# B&R Automation Studio project EFI (part 7)

### IOMap.iom - PC_any/IOMap.iom
```iecst
(********************************************************************
 * COPYRIGHT -- Bernecker + Rainer
 ********************************************************************
 * File: IoMap.iom
 * Author: B+R
 ********************************************************************
 * IO mapping file
 ********************************************************************)
VAR_CONFIG
	Cyclic#1.::gAxisStepper[1].DrvIf.iLifeCnt AT %IB."X67SM2436".LifeCnt;
	Cyclic#1.::gAxisStepper[1].DrvIf.iDrvOK AT %IX."X67SM2436".DrvOk01;
	Cyclic#1.::gAxisStepper[1].DrvIf.oBoostCurrent AT %QX."X67SM2436".BoostCurrent01;
	Cyclic#1.::gAxisStepper[1].DrvIf.oStandStillCurrent AT %QX."X67SM2436".StandstillCurrent01;
	Cyclic#1.::gAxisStepper[1].DrvIf.oSetTime AT %QW."X67SM2436".SetTime01;
	Cyclic#1.::gAxisStepper[1].MotorStep0 AT %QW."X67SM2436".Motor1Step0;
	Cyclic#1.::gAxisStepper[1].DiDoIf.iLifeCntDriveEnable AT %IB."X67SM2436".LifeCnt;
	Cyclic#1.::gAxisStepper[1].DiDoIf.iLifeCntDriveReady AT %IB."X67SM2436".LifeCnt;
	Cyclic#1.::gAxisStepper[1].DiDoIf.iDriveReady AT %IX."X67SM2436".DrvOk01;
	Cyclic#1.::gAxisStepper[1].DiDoIf.oDriveEnable AT %QX."X67SM2436".DriveEnable01;
	Cyclic#1.::gAxisStepper[1].EncIf1.iLifeCnt AT %IB."X67SM2436".LifeCnt;
	Cyclic#1.::gAxisStepper[1].EncIf1.iEncOK AT %IX."X67SM2436".EncOk01;
	Cyclic#1.::gAxisStepper[1].EncIf1.iActPos AT %IW."X67SM2436".ActPos01;
	Cyclic#1.::gAxisStepper[1].EncIf1.iRefPulsePos AT %IW."X67SM2436".RefPulsePos01;
	Cyclic#1.::gAxisStepper[1].EncIf1.iRefPulseCnt AT %IB."X67SM2436".RefPulseCnt01;
	Cyclic#1.::gAxisStepper[1].EncIf1.iActTime AT %IW."X67SM2436".ActTime01;
	Cyclic#1.::gAxisStepper[2].DrvIf.iLifeCnt AT %IB."X67SM2436".LifeCnt;
	Cyclic#1.::gAxisStepper[2].DrvIf.iDrvOK AT %IX."X67SM2436".DrvOk02;
	Cyclic#1.::gAxisStepper[2].DrvIf.oBoostCurrent AT %QX."X67SM2436".BoostCurrent02;
	Cyclic#1.::gAxisStepper[2].DrvIf.oStandStillCurrent AT %QX."X67SM2436".StandstillCurrent02;
	Cyclic#1.::gAxisStepper[2].DrvIf.oSetTime AT %QW."X67SM2436".SetTime02;
	Cyclic#1.::gAxisStepper[2].MotorStep0 AT %QW."X67SM2436".Motor2Step0;
	Cyclic#1.::gAxisStepper[2].DiDoIf.iLifeCntDriveEnable AT %IB."X67SM2436".LifeCnt;
	Cyclic#1.::gAxisStepper[2].DiDoIf.iLifeCntDriveReady AT %IB."X67SM2436".LifeCnt;
	Cyclic#1.::gAxisStepper[2].DiDoIf.iDriveReady AT %IX."X67SM2436".DrvOk02;
	Cyclic#1.::gAxisStepper[2].DiDoIf.oDriveEnable AT %QX."X67SM2436".DriveEnable02;
	Cyclic#1.::gAxisStepper[2].EncIf1.iLifeCnt AT %IB."X67SM2436".LifeCnt;
	Cyclic#1.::gAxisStepper[2].EncIf1.iEncOK AT %IX."X67SM2436".EncOk02;
	Cyclic#1.::gAxisStepper[2].EncIf1.iActPos AT %IW."X67SM2436".ActPos02;
	Cyclic#1.::gAxisStepper[2].EncIf1.iRefPulsePos AT %IW."X67SM2436".RefPulsePos02;
	Cyclic#1.::gAxisStepper[2].EncIf1.iRefPulseCnt AT %IB."X67SM2436".RefPulseCnt02;
	Cyclic#1.::gAxisStepper[2].EncIf1.iActTime AT %IW."X67SM2436".ActTime02;
	Cyclic#1.::gInverterSignalsPowerLink[1].In.StatusWord AT %IW."8I66xxxxxxx.0P-xxx1".ETAD_Input;
	Cyclic#1.::gInverterSignalsPowerLink[1].In.ActualSpeed AT %IW."8I66xxxxxxx.0P-xxx1".RFRD_Input;
	Cyclic#1.::gInverterSignalsPowerLink[1].In.ErrorID AT %IW."8I66xxxxxxx.0P-xxx1".LFT_Input;
	Cyclic#1.::gInverterSignalsPowerLink[1].Out.ControlWord AT %QW."8I66xxxxxxx.0P-xxx1".CMDD_Output;
	Cyclic#1.::gInverterSignalsPowerLink[1].Out.SetSpeed AT %QW."8I66xxxxxxx.0P-xxx1".LFRD_Output;
	Cyclic#1.::gInverterSignalsPowerLink[1].In.ActualCurrent AT %IW."8I66xxxxxxx.0P-xxx1".LCR_Input;
	Cyclic#1.::gInverterSignalsPowerLink[1].In.DigitalInput[0] AT %IX."8I66xxxxxxx.0P-xxx1".IL1R_Input_DI1;
	Cyclic#1.::gInverterSignalsPowerLink[1].In.DigitalInput[1] AT %IX."8I66xxxxxxx.0P-xxx1".IL1R_Input_DI2;
	Cyclic#1.::gInverterSignalsPowerLink[1].In.DigitalInput[2] AT %IX."8I66xxxxxxx.0P-xxx1".IL1R_Input_DI3;
	Cyclic#1.::gInverterSignalsPowerLink[1].In.DigitalInput[3] AT %IX."8I66xxxxxxx.0P-xxx1".IL1R_Input_DI4;
	Cyclic#1.::gInverterSignalsPowerLink[1].In.DigitalInput[4] AT %IX."8I66xxxxxxx.0P-xxx1".IL1R_Input_DI5;
	Cyclic#1.::gInverterSignalsPowerLink[1].In.DigitalInput[5] AT %IX."8I66xxxxxxx.0P-xxx1".IL1R_Input_DI6;
	Cyclic#1.::gInverterSignalsPowerLink[1].In.DigitalInput[6] AT %IX."8I66xxxxxxx.0P-xxx1".IL1R_Input_DAI1;
	Cyclic#1.::gInverterSignalsPowerLink[1].In.DigitalInput[7] AT %IX."8I66xxxxxxx.0P-xxx1".IL1R_Input_DAI2;
	Cyclic#1.::gInverterSignalsPowerLink[1].In.AnalogInput[0] AT %IW."8I66xxxxxxx.0P-xxx1".AI1R_Input;
	Cyclic#1.::gInverterSignalsPowerLink[1].In.AnalogInput[1] AT %IW."8I66xxxxxxx.0P-xxx1".AI2R_Input;
	Cyclic#1.::gInverterSignalsPowerLink[1].In.AnalogInput[2] AT %IW."8I66xxxxxxx.0P-xxx1".AI3R_Input;
	Cyclic#1.::gInverterSignalsPowerLink[1].Out.AnalogOutput AT %QW."8I66xxxxxxx.0P-xxx1".AO1R_Output;
	Cyclic#1.::gInverterSignalsPowerLink[1].Out.DigitalOutput[0] AT %QX."8I66xxxxxxx.0P-xxx1".OL1R_Output_R1;
	Cyclic#1.::gInverterSignalsPowerLink[1].Out.DigitalOutput[1] AT %QX."8I66xxxxxxx.0P-xxx1".OL1R_Output_R2;
	Cyclic#1.::gInverterSignalsPowerLink[1].Out.DigitalOutput[2] AT %QX."8I66xxxxxxx.0P-xxx1".OL1R_Output_DQ1;
	Cyclic#1.::gInverterSignalsPowerLink[1].In.ActualTorque AT %IW."8I66xxxxxxx.0P-xxx1".OTRN_Input;
	gToWriteDataModbFeeder[1] AT %QW."ModbusFeeder".writeFeederBk2_1;
	gToWriteDataModbFeeder[2] AT %QW."ModbusFeeder".writeFeederBk2_2;
	gToWriteDataModbFeeder[3] AT %QW."ModbusFeeder".writeFeederBk2_3;
	gToWriteDataModbFeeder[4] AT %QW."ModbusFeeder".writeFeederBk2_4;
	gToWriteDataModbFeeder[5] AT %QX."ModbusFeeder".writeFeederBk2_5;
	gToWriteDataModbFeeder[6] AT %QX."ModbusFeeder".writeFeederBk2_6;
	gToWriteDataModbFeeder[7] AT %QX."ModbusFeeder".writeFeederBk2_7;
	gToWriteDataModbFeeder[8] AT %QX."ModbusFeeder".writeFeederBk2_8;
	gToWriteDataModbFeeder[9] AT %QX."ModbusFeeder".writeFeederBk2_9;
	gToWriteDataModbFeeder[10] AT %QX."ModbusFeeder".writeFeederBk2_10;
	gToWriteDataModbFeeder[11] AT %QX."ModbusFeeder".writeFeederBk2_11;
	gToWriteDataModbFeeder[12] AT %QX."ModbusFeeder".writeFeederBk2_12;
	gToWriteDataModbFeeder[13] AT %QX."ModbusFeeder".writeFeederBk2_13;
	gToWriteDataModbFeeder[14] AT %QX."ModbusFeeder".writeFeederBk2_14;
	gToWriteDataModbFeeder[15] AT %QX."ModbusFeeder".writeFeederBk2_15;
	gToWriteDataModbFeeder[16] AT %QX."ModbusFeeder".writeFeederBk2_16;
	gToWriteDataModbFeeder[17] AT %QX."ModbusFeeder".writeFeederBk2_17;
	gToWriteDataModbFeeder[18] AT %QX."ModbusFeeder".writeFeederBk2_18;
	gToWriteDataModbFeeder[19] AT %QX."ModbusFeeder".writeFeederBk2_19;
	gToWriteDataModbFeeder[20] AT %QX."ModbusFeeder".writeFeederBk2_20;
	gToWriteDataModbFeeder[21] AT %QX."ModbusFeeder".writeFeederBk2_21;
	gToWriteDataModbFeeder[22] AT %QX."ModbusFeeder".writeFeederBk2_22;
	gToWriteDataModbFeeder[23] AT %QX."ModbusFeeder".writeFeederBk2_23;
	gToWriteDataModbFeeder[24] AT %QX."ModbusFeeder".writeFeederBk2_24;
	gToWriteDataModbFeeder[25] AT %QX."ModbusFeeder".writeFeederBk2_25;
	gReceivedDataModbFeeder[1] AT %IW."ModbusFeeder".readFeederBk1_1;
	gReceivedDataModbFeeder[2] AT %IW."ModbusFeeder".readFeederBk1_2;
	gReceivedDataModbFeeder[3] AT %IW."ModbusFeeder".readFeederBk1_3;
	gReceivedDataModbFeeder[4] AT %IW."ModbusFeeder".readFeederBk1_4;
	gToWriteDataModbFeeder[5] AT %IX."ModbusFeeder".readFeederBk1_5;
	gToWriteDataModbFeeder[6] AT %IX."ModbusFeeder".readFeederBk1_6;
	gToWriteDataModbFeeder[7] AT %IX."ModbusFeeder".readFeederBk1_7;
	gToWriteDataModbFeeder[8] AT %IX."ModbusFeeder".readFeederBk1_8;
	gToWriteDataModbFeeder[9] AT %IX."ModbusFeeder".readFeederBk1_9;
	gToWriteDataModbFeeder[10] AT %IX."ModbusFeeder".readFeederBk1_10;
	gToWriteDataModbFeeder[11] AT %IX."ModbusFeeder".readFeederBk1_11;
	gToWriteDataModbFeeder[12] AT %IX."ModbusFeeder".readFeederBk1_12;
	gToWriteDataModbFeeder[13] AT %IX."ModbusFeeder".readFeederBk1_13;
	gToWriteDataModbFeeder[14] AT %IX."ModbusFeeder".readFeederBk1_14;
	gToWriteDataModbFeeder[15] AT %IX."ModbusFeeder".readFeederBk1_15;
	gToWriteDataModbFeeder[16] AT %IX."ModbusFeeder".readFeederBk1_16;
	gToWriteDataModbFeeder[17] AT %IX."ModbusFeeder".readFeederBk1_17;
	gToWriteDataModbFeeder[18] AT %IX."ModbusFeeder".readFeederBk1_18;
	gToWriteDataModbFeeder[19] AT %IX."ModbusFeeder".readFeederBk1_19;
	gToWriteDataModbFeeder[20] AT %IX."ModbusFeeder".readFeederBk1_20;
	gToWriteDataModbFeeder[21] AT %IX."ModbusFeeder".readFeederBk1_21;
	gToWriteDataModbFeeder[22] AT %IX."ModbusFeeder".readFeederBk1_22;
	gToWriteDataModbFeeder[23] AT %IX."ModbusFeeder".readFeederBk1_23;
	gToWriteDataModbFeeder[24] AT %IX."ModbusFeeder".readFeederBk1_24;
	gToWriteDataModbFeeder[25] AT %IX."ModbusFeeder".readFeederBk1_25;
	gToWriteDataModbCoater[1] AT %QW."ModbusPrimer".writeCoaterBk2_1;
	gToWriteDataModbCoater[2] AT %QW."ModbusPrimer".writeCoaterBk2_2;
	gToWriteDataModbCoater[3] AT %QW."ModbusPrimer".writeCoaterBk2_3;
	gToWriteDataModbCoater[4] AT %QW."ModbusPrimer".writeCoaterBk2_4;
	gToWriteDataModbCoater[5] AT %QW."ModbusPrimer".writeCoaterBk2_5;
	gToWriteDataModbCoater[6] AT %QW."ModbusPrimer".writeCoaterBk2_6;
	gToWriteDataModbCoater[7] AT %QW."ModbusPrimer".writeCoaterBk2_7;
	gToWriteDataModbCoater[8] AT %QW."ModbusPrimer".writeCoaterBk2_8;
	gToWriteDataModbCoater[9] AT %QW."ModbusPrimer".writeCoaterBk2_9;
	gToWriteDataModbCoater[10] AT %QW."ModbusPrimer".writeCoaterBk2_10;
	gToWriteDataModbCoater[11] AT %QW."ModbusPrimer".writeCoaterBk2_11;
	gToWriteDataModbCoater[12] AT %QW."ModbusPrimer".writeCoaterBk2_12;
	gToWriteDataModbCoater[13] AT %QW."ModbusPrimer".writeCoaterBk2_13;
	gToWriteDataModbCoater[14] AT %QW."ModbusPrimer".writeCoaterBk2_14;
	gToWriteDataModbCoater[15] AT %QW."ModbusPrimer".writeCoaterBk2_15;
	gToWriteDataModbCoater[16] AT %QW."ModbusPrimer".writeCoaterBk2_16;
	gToWriteDataModbCoater[17] AT %QW."ModbusPrimer".writeCoaterBk2_17;
	gToWriteDataModbCoater[18] AT %QW."ModbusPrimer".writeCoaterBk2_18;
	gToWriteDataModbCoater[19] AT %QW."ModbusPrimer".writeCoaterBk2_19;
	gToWriteDataModbCoater[20] AT %QW."ModbusPrimer".writeCoaterBk2_20;
	gToWriteDataModbCoater[21] AT %QW."ModbusPrimer".writeCoaterBk2_21;
	gToWriteDataModbCoater[22] AT %QW."ModbusPrimer".writeCoaterBk2_22;
	gToWriteDataModbCoater[23] AT %QW."ModbusPrimer".writeCoaterBk2_23;
	gToWriteDataModbCoater[24] AT %QW."ModbusPrimer".writeCoaterBk2_24;
	gToWriteDataModbCoater[25] AT %QW."ModbusPrimer".writeCoaterBk2_25;
	gReceivedDataModbCoater[1] AT %QW."ModbusPrimer".readCoaterBk1_1;
	gReceivedDataModbCoater[2] AT %QW."ModbusPrimer".readCoaterBk1_2;
	gReceivedDataModbCoater[3] AT %QW."ModbusPrimer".readCoaterBk1_3;
	gReceivedDataModbCoater[4] AT %QW."ModbusPrimer".readCoaterBk1_4;
	gReceivedDataModbCoater[5] AT %QW."ModbusPrimer".readCoaterBk1_5;
	gReceivedDataModbCoater[6] AT %QW."ModbusPrimer".readCoaterBk1_6;
	gReceivedDataModbCoater[7] AT %QW."ModbusPrimer".readCoaterBk1_7;
	gReceivedDataModbCoater[8] AT %QW."ModbusPrimer".readCoaterBk1_8;
	gReceivedDataModbCoater[9] AT %QW."ModbusPrimer".readCoaterBk1_9;
	gReceivedDataModbCoater[10] AT %QW."ModbusPrimer".readCoaterBk1_10;
	gReceivedDataModbCoater[11] AT %QW."ModbusPrimer".readCoaterBk1_11;
	gReceivedDataModbCoater[12] AT %QW."ModbusPrimer".readCoaterBk1_12;
	gReceivedDataModbCoater[13] AT %QW."ModbusPrimer".readCoaterBk1_13;
	gReceivedDataModbCoater[14] AT %QW."ModbusPrimer".readCoaterBk1_14;
	gReceivedDataModbCoater[15] AT %QW."ModbusPrimer".readCoaterBk1_15;
	gReceivedDataModbCoater[16] AT %QW."ModbusPrimer".readCoaterBk1_16;
	gReceivedDataModbCoater[17] AT %QW."ModbusPrimer".readCoaterBk1_17;
	gReceivedDataModbCoater[18] AT %QW."ModbusPrimer".readCoaterBk1_18;
	gReceivedDataModbCoater[19] AT %QW."ModbusPrimer".readCoaterBk1_19;
	gReceivedDataModbCoater[20] AT %QW."ModbusPrimer".readCoaterBk1_20;
	gReceivedDataModbCoater[21] AT %QW."ModbusPrimer".readCoaterBk1_21;
	gReceivedDataModbCoater[22] AT %QW."ModbusPrimer".readCoaterBk1_22;
	gReceivedDataModbCoater[23] AT %QW."ModbusPrimer".readCoaterBk1_23;
	gReceivedDataModbCoater[24] AT %QW."ModbusPrimer".readCoaterBk1_24;
	gReceivedDataModbCoater[25] AT %QW."ModbusPrimer".readCoaterBk1_25;
	gReceivedDataModbFeeder[5] AT %IW."ModbusFeeder".readFeederBk1_5;
	gReceivedDataModbFeeder[6] AT %IW."ModbusFeeder".readFeederBk1_6;
	gReceivedDataModbFeeder[7] AT %IW."ModbusFeeder".readFeederBk1_7;
	gReceivedDataModbFeeder[8] AT %IW."ModbusFeeder".readFeederBk1_8;
	gReceivedDataModbFeeder[9] AT %IW."ModbusFeeder".readFeederBk1_9;
	gReceivedDataModbFeeder[10] AT %IW."ModbusFeeder".readFeederBk1_10;
	gReceivedDataModbFeeder[11] AT %IW."ModbusFeeder".readFeederBk1_11;
	gReceivedDataModbFeeder[12] AT %IW."ModbusFeeder".readFeederBk1_12;
	gReceivedDataModbFeeder[13] AT %IW."ModbusFeeder".readFeederBk1_13;
	gReceivedDataModbFeeder[14] AT %IW."ModbusFeeder".readFeederBk1_14;
	gReceivedDataModbFeeder[15] AT %IW."ModbusFeeder".readFeederBk1_15;
	gReceivedDataModbFeeder[16] AT %IW."ModbusFeeder".readFeederBk1_16;
	gReceivedDataModbFeeder[17] AT %IW."ModbusFeeder".readFeederBk1_17;
	gReceivedDataModbFeeder[18] AT %IW."ModbusFeeder".readFeederBk1_18;
	gReceivedDataModbFeeder[19] AT %IW."ModbusFeeder".readFeederBk1_19;
	gReceivedDataModbFeeder[20] AT %IW."ModbusFeeder".readFeederBk1_20;
	gReceivedDataModbFeeder[21] AT %IW."ModbusFeeder".readFeederBk1_21;
	gReceivedDataModbFeeder[22] AT %IW."ModbusFeeder".readFeederBk1_22;
	gReceivedDataModbFeeder[23] AT %IW."ModbusFeeder".readFeederBk1_23;
	gReceivedDataModbFeeder[24] AT %IW."ModbusFeeder".readFeederBk1_24;
	gReceivedDataModbFeeder[25] AT %IW."ModbusFeeder".readFeederBk1_25;
	gToWriteDataModbFeeder[5] AT %QW."ModbusFeeder".writeFeederBk2_5;
	gToWriteDataModbFeeder[6] AT %QW."ModbusFeeder".writeFeederBk2_6;
	gToWriteDataModbFeeder[7] AT %QW."ModbusFeeder".writeFeederBk2_7;
	gToWriteDataModbFeeder[8] AT %QW."ModbusFeeder".writeFeederBk2_8;
	gToWriteDataModbFeeder[9] AT %QW."ModbusFeeder".writeFeederBk2_9;
	gToWriteDataModbFeeder[10] AT %QW."ModbusFeeder".writeFeederBk2_10;
	gToWriteDataModbFeeder[11] AT %QW."ModbusFeeder".writeFeederBk2_11;
	gToWriteDataModbFeeder[12] AT %QW."ModbusFeeder".writeFeederBk2_12;
	gToWriteDataModbFeeder[13] AT %QW."ModbusFeeder".writeFeederBk2_13;
	gToWriteDataModbFeeder[14] AT %QW."ModbusFeeder".writeFeederBk2_14;
	gToWriteDataModbFeeder[15] AT %QW."ModbusFeeder".writeFeederBk2_15;
	gToWriteDataModbFeeder[16] AT %QW."ModbusFeeder".writeFeederBk2_16;
	gToWriteDataModbFeeder[17] AT %QW."ModbusFeeder".writeFeederBk2_17;
	gToWriteDataModbFeeder[18] AT %QW."ModbusFeeder".writeFeederBk2_18;
	gToWriteDataModbFeeder[19] AT %QW."ModbusFeeder".writeFeederBk2_19;
	gToWriteDataModbFeeder[20] AT %QW."ModbusFeeder".writeFeederBk2_20;
	gToWriteDataModbFeeder[21] AT %QW."ModbusFeeder".writeFeederBk2_21;
	gToWriteDataModbFeeder[22] AT %QW."ModbusFeeder".writeFeederBk2_22;
	gToWriteDataModbFeeder[23] AT %QW."ModbusFeeder".writeFeederBk2_23;
	gToWriteDataModbFeeder[24] AT %QW."ModbusFeeder".writeFeederBk2_24;
	gToWriteDataModbFeeder[25] AT %QW."ModbusFeeder".writeFeederBk2_25;
	gReceivedDataModbCoater[1] AT %IW."ModbusPrimer".readCoaterBk1_1;
	gReceivedDataModbCoater[2] AT %IW."ModbusPrimer".readCoaterBk1_2;
	gReceivedDataModbCoater[3] AT %IW."ModbusPrimer".readCoaterBk1_3;
	gReceivedDataModbCoater[4] AT %IW."ModbusPrimer".readCoaterBk1_4;
	gReceivedDataModbCoater[5] AT %IW."ModbusPrimer".readCoaterBk1_5;
	gReceivedDataModbCoater[6] AT %IW."ModbusPrimer".readCoaterBk1_6;
	gReceivedDataModbCoater[7] AT %IW."ModbusPrimer".readCoaterBk1_7;
	gReceivedDataModbCoater[8] AT %IW."ModbusPrimer".readCoaterBk1_8;
	gReceivedDataModbCoater[9] AT %IW."ModbusPrimer".readCoaterBk1_9;
	gReceivedDataModbCoater[10] AT %IW."ModbusPrimer".readCoaterBk1_10;
	gReceivedDataModbCoater[11] AT %IW."ModbusPrimer".readCoaterBk1_11;
	gReceivedDataModbCoater[12] AT %IW."ModbusPrimer".readCoaterBk1_12;
	gReceivedDataModbCoater[13] AT %IW."ModbusPrimer".readCoaterBk1_13;
	gReceivedDataModbCoater[14] AT %IW."ModbusPrimer".readCoaterBk1_14;
	gReceivedDataModbCoater[15] AT %IW."ModbusPrimer".readCoaterBk1_15;
	gReceivedDataModbCoater[16] AT %IW."ModbusPrimer".readCoaterBk1_16;
	gReceivedDataModbCoater[17] AT %IW."ModbusPrimer".readCoaterBk1_17;
	gReceivedDataModbCoater[18] AT %IW."ModbusPrimer".readCoaterBk1_18;
	gReceivedDataModbCoater[19] AT %IW."ModbusPrimer".readCoaterBk1_19;
	gReceivedDataModbCoater[20] AT %IW."ModbusPrimer".readCoaterBk1_20;
	gReceivedDataModbCoater[21] AT %IW."ModbusPrimer".readCoaterBk1_21;
	gReceivedDataModbCoater[22] AT %IW."ModbusPrimer".readCoaterBk1_22;
	gReceivedDataModbCoater[23] AT %IW."ModbusPrimer".readCoaterBk1_23;
	gReceivedDataModbCoater[24] AT %IW."ModbusPrimer".readCoaterBk1_24;
	gReceivedDataModbCoater[25] AT %IW."ModbusPrimer".readCoaterBk1_25;
	gReceivedDataModbSafety[1] AT %IW."ModbusSafety".readSafetyBk1_1;
	gReceivedDataModbSafety[2] AT %IW."ModbusSafety".readSafetyBk1_2;
	gReceivedDataModbSafety[3] AT %IW."ModbusSafety".readSafetyBk1_3;
	gReceivedDataModbSafety[4] AT %IW."ModbusSafety".readSafetyBk1_4;
	gReceivedDataModbSafety[5] AT %IW."ModbusSafety".readSafetyBk1_5;
	gReceivedDataModbSafety[6] AT %IW."ModbusSafety".readSafetyBk1_6;
	gReceivedDataModbSafety[7] AT %IW."ModbusSafety".readSafetyBk1_7;
	gReceivedDataModbSafety[8] AT %IW."ModbusSafety".readSafetyBk1_8;
	gReceivedDataModbSafety[9] AT %IW."ModbusSafety".readSafetyBk1_9;
	gReceivedDataModbSafety[10] AT %IW."ModbusSafety".readSafetyBk1_10;
	gReceivedDataModbSafety[11] AT %IW."ModbusSafety".readSafetyBk1_11;
	gReceivedDataModbSafety[12] AT %IW."ModbusSafety".readSafetyBk1_12;
	gToWriteDataModbSafety AT %QW."ModbusSafety".writeSafetyBk2_1;
	gReceivedDataModbStacker[1] AT %IW."ModbusStacker".readStackerBk1_1;
	gReceivedDataModbStacker[2] AT %IW."ModbusStacker".readStackerBk1_2;
	gReceivedDataModbStacker[3] AT %IW."ModbusStacker".readStackerBk1_3;
	gReceivedDataModbStacker[4] AT %IW."ModbusStacker".readStackerBk1_4;
	gReceivedDataModbStacker[5] AT %IW."ModbusStacker".readStackerBk1_5;
	gReceivedDataModbStacker[6] AT %IW."ModbusStacker".readStackerBk1_6;
	gReceivedDataModbStacker[7] AT %IW."ModbusStacker".readStackerBk1_7;
	gReceivedDataModbStacker[8] AT %IW."ModbusStacker".readStackerBk1_8;
	gReceivedDataModbStacker[9] AT %IW."ModbusStacker".readStackerBk1_9;
	gReceivedDataModbStacker[10] AT %IW."ModbusStacker".readStackerBk1_10;
	gReceivedDataModbStacker[11] AT %IW."ModbusStacker".readStackerBk1_11;
	gReceivedDataModbStacker[12] AT %IW."ModbusStacker".readStackerBk1_12;
	gReceivedDataModbStacker[13] AT %IW."ModbusStacker".readStackerBk1_13;
	gReceivedDataModbStacker[14] AT %IW."ModbusStacker".readStackerBk1_14;
	gReceivedDataModbStacker[15] AT %IW."ModbusStacker".readStackerBk1_15;
	gReceivedDataModbStacker[16] AT %IW."ModbusStacker".readStackerBk1_16;
	gReceivedDataModbStacker[17] AT %IW."ModbusStacker".readStackerBk1_17;
	gReceivedDataModbStacker[18] AT %IW."ModbusStacker".readStackerBk1_18;
	gReceivedDataModbStacker[19] AT %IW."ModbusStacker".readStackerBk1_19;
	gReceivedDataModbStacker[20] AT %IW."ModbusStacker".readStackerBk1_20;
	gReceivedDataModbStacker[21] AT %IW."ModbusStacker".readStackerBk1_21;
	gReceivedDataModbStacker[22] AT %IW."ModbusStacker".readStackerBk1_22;
	gReceivedDataModbStacker[23] AT %IW."ModbusStacker".readStackerBk1_23;
	gReceivedDataModbStacker[24] AT %IW."ModbusStacker".readStackerBk1_24;
	gReceivedDataModbStacker[25] AT %IW."ModbusStacker".readStackerBk1_25;
	gToWriteDataModbStacker[1] AT %QW."ModbusStacker".writeStackerBk2_1;
	gToWriteDataModbStacker[2] AT %QW."ModbusStacker".writeStackerBk2_2;
	gToWriteDataModbStacker[3] AT %QW."ModbusStacker".writeStackerBk2_3;
	gToWriteDataModbStacker[4] AT %QW."ModbusStacker".writeStackerBk2_4;
	gToWriteDataModbStacker[5] AT %QW."ModbusStacker".writeStackerBk2_5;
	gToWriteDataModbStacker[6] AT %QW."ModbusStacker".writeStackerBk2_6;
	gToWriteDataModbStacker[7] AT %QW."ModbusStacker".writeStackerBk2_7;
	gToWriteDataModbStacker[8] AT %QW."ModbusStacker".writeStackerBk2_8;
	gToWriteDataModbStacker[9] AT %QW."ModbusStacker".writeStackerBk2_9;
	gToWriteDataModbStacker[10] AT %QW."ModbusStacker".writeStackerBk2_10;
	gToWriteDataModbStacker[11] AT %QW."ModbusStacker".writeStackerBk2_11;
	gToWriteDataModbStacker[12] AT %QW."ModbusStacker".writeStackerBk2_12;
	gToWriteDataModbStacker[13] AT %QW."ModbusStacker".writeStackerBk2_13;
	gToWriteDataModbStacker[14] AT %QW."ModbusStacker".writeStackerBk2_14;
	gToWriteDataModbStacker[15] AT %QW."ModbusStacker".writeStackerBk2_15;
	gToWriteDataModbStacker[16] AT %QW."ModbusStacker".writeStackerBk2_16;
	gToWriteDataModbStacker[17] AT %QW."ModbusStacker".writeStackerBk2_17;
	gToWriteDataModbStacker[18] AT %QW."ModbusStacker".writeStackerBk2_18;
	gToWriteDataModbStacker[19] AT %QW."ModbusStacker".writeStackerBk2_19;
	gToWriteDataModbStacker[20] AT %QW."ModbusStacker".writeStackerBk2_20;
	gToWriteDataModbStacker[21] AT %QW."ModbusStacker".writeStackerBk2_21;
	gToWriteDataModbStacker[22] AT %QW."ModbusStacker".writeStackerBk2_22;
	gToWriteDataModbStacker[23] AT %QW."ModbusStacker".writeStackerBk2_23;
	gToWriteDataModbStacker[24] AT %QW."ModbusStacker".writeStackerBk2_24;
	gToWriteDataModbStacker[25] AT %QW."ModbusStacker".writeStackerBk2_25;
	gReceivedDataModPowerMeter1[1] AT %IX."ModbusPowerMeter".readPowerMeterBk1_1;
	gReceivedDataModPowerMeter1[16] AT %IX."ModbusPowerMeter".readPowerMeterBk2_1;
	gReceivedDataModPowerMeter1[1] AT %IW."ModbusPowerMeter".readPowerMeterBk1_1;
	gReceivedDataModPowerMeter1[2] AT %IW."ModbusPowerMeter".readPowerMeterBk1_2;
	gReceivedDataModPowerMeter1[3] AT %IW."ModbusPowerMeter".readPowerMeterBk1_3;
	gReceivedDataModPowerMeter1[4] AT %IW."ModbusPowerMeter".readPowerMeterBk1_4;
	gReceivedDataModPowerMeter1[5] AT %IX."ModbusPowerMeter".readPowerMeterBk1_5;
	gReceivedDataModPowerMeter1[6] AT %IX."ModbusPowerMeter".readPowerMeterBk1_6;
	gReceivedDataModPowerMeter1[16] AT %IW."ModbusPowerMeter".readPowerMeterBk2_1;
	gReceivedDataModPowerMeter1[36] AT %IX."ModbusPowerMeter".readPowerMeterBk2_2;
	gReceivedDataModPowerMeter1[18] AT %IW."ModbusPowerMeter".readPowerMeterBk2_3;
	gReceivedDataModPowerMeter1[19] AT %IW."ModbusPowerMeter".readPowerMeterBk2_4;
	gReceivedDataModPowerMeter1[20] AT %IW."ModbusPowerMeter".readPowerMeterBk2_5;
	gReceivedDataModPowerMeter1[21] AT %IW."ModbusPowerMeter".readPowerMeterBk2_6;
	gReceivedDataModPowerMeter1[22] AT %IW."ModbusPowerMeter".readPowerMeterBk2_7;
	gReceivedDataModPowerMeter1[23] AT %IW."ModbusPowerMeter".readPowerMeterBk2_8;
	gReceivedDataModPowerMeter1[24] AT %IW."ModbusPowerMeter".readPowerMeterBk2_9;
	gReceivedDataModPowerMeter1[25] AT %IW."ModbusPowerMeter".readPowerMeterBk2_10;
	gReceivedDataModPowerMeter1[26] AT %IW."ModbusPowerMeter".readPowerMeterBk2_11;
	gReceivedDataModPowerMeter1[27] AT %IW."ModbusPowerMeter".readPowerMeterBk2_12;
	gReceivedDataModPowerMeter1[28] AT %IW."ModbusPowerMeter".readPowerMeterBk2_13;
	gReceivedDataModPowerMeter1[29] AT %IW."ModbusPowerMeter".readPowerMeterBk2_14;
	gReceivedDataModPowerMeter1[30] AT %IW."ModbusPowerMeter".readPowerMeterBk2_15;
	gReceivedDataModPowerMeter1[31] AT %IW."ModbusPowerMeter".readPowerMeterBk2_16;
	gReceivedDataModPowerMeter1[32] AT %IW."ModbusPowerMeter".readPowerMeterBk2_17;
	gReceivedDataModPowerMeter1[33] AT %IW."ModbusPowerMeter".readPowerMeterBk2_18;
	gReceivedDataModPowerMeter1[34] AT %IW."ModbusPowerMeter".readPowerMeterBk2_19;
	gReceivedDataModPowerMeter1[35] AT %IW."ModbusPowerMeter".readPowerMeterBk2_20;
	gReceivedDataModPowerMeter1[36] AT %IW."ModbusPowerMeter".readPowerMeterBk2_21;
	gReceivedDataModPowerMeter1[37] AT %IW."ModbusPowerMeter".readPowerMeterBk2_22;
	gReceivedDataModPowerMeter1[38] AT %IW."ModbusPowerMeter".readPowerMeterBk2_23;
	gReceivedDataModPowerMeter1[39] AT %IW."ModbusPowerMeter".readPowerMeterBk2_24;
	gReceivedDataModPowerMeter1[40] AT %IW."ModbusPowerMeter".readPowerMeterBk2_25;
	gReceivedDataModPowerMeter1[41] AT %IW."ModbusPowerMeter".readPowerMeterBk2_26;
	gReceivedDataModPowerMeter1[42] AT %IW."ModbusPowerMeter".readPowerMeterBk2_27;
	gReceivedDataModPowerMeter1[43] AT %IW."ModbusPowerMeter".readPowerMeterBk2_28;
	gReceivedDataModPowerMeter1[44] AT %IW."ModbusPowerMeter".readPowerMeterBk2_29;
	gReceivedDataModPowerMeter1[45] AT %IW."ModbusPowerMeter".readPowerMeterBk2_30;
	gReceivedDataModPowerMeter1[46] AT %IW."ModbusPowerMeter".readPowerMeterBk2_31;
	gReceivedDataModPowerMeter1[47] AT %IW."ModbusPowerMeter".readPowerMeterBk2_32;
	gReceivedDataModPowerMeter1[48] AT %IW."ModbusPowerMeter".readPowerMeterBk2_33;
	gReceivedDataModPowerMeter1[49] AT %IW."ModbusPowerMeter".readPowerMeterBk2_34;
	gReceivedDataModPowerMeter1[50] AT %IW."ModbusPowerMeter".readPowerMeterBk2_35;
	gReceivedDataModPowerMeter1[104] AT %IW."ModbusPowerMeter".readPowerMeterBk3_1;
	gReceivedDataModPowerMeter1[105] AT %IW."ModbusPowerMeter".readPowerMeterBk3_2;
	gReceivedDataModPowerMeter1[106] AT %IW."ModbusPowerMeter".readPowerMeterBk3_3;
	gReceivedDataModPowerMeter1[107] AT %IW."ModbusPowerMeter".readPowerMeterBk3_4;
	gReceivedDataModPowerMeter1[108] AT %IW."ModbusPowerMeter".readPowerMeterBk3_5;
	gReceivedDataModPowerMeter1[109] AT %IW."ModbusPowerMeter".readPowerMeterBk3_6;
	gReceivedDataModPowerMeter1[110] AT %IW."ModbusPowerMeter".readPowerMeterBk3_7;
	gReceivedDataModPowerMeter1[111] AT %IW."ModbusPowerMeter".readPowerMeterBk3_8;
	gReceivedDataModPowerMeter1[112] AT %IW."ModbusPowerMeter".readPowerMeterBk3_9;
	gReceivedDataModPowerMeter1[113] AT %IW."ModbusPowerMeter".readPowerMeterBk3_10;
	gReceivedDataModPowerMeter1[5] AT %IW."ModbusPowerMeter".readPowerMeterBk1_5;
	gReceivedDataModPowerMeter1[6] AT %IW."ModbusPowerMeter".readPowerMeterBk1_6;
	gReceivedDataModPowerMeter1[17] AT %IW."ModbusPowerMeter".readPowerMeterBk2_2;
	::gDryerAnc.Inputs.xTransportMoving AT %IX."OpcUaDryer".xRuningBelt;
	::gDryerAnc.Outputs.xRunTransport AT %QX."OpcUaDryer".xRunTransport;
	::gDryerAnc.Outputs.xPrepareToDry AT %QX."OpcUaDryer".xPrepareToDry;
	::gDryerAnc.Outputs.xStartDrying AT %QX."OpcUaDryer".xStartDrying;
	::gDryerAnc.Inputs.xDrying AT %IX."OpcUaDryer".xDrying;
	::gDryerAnc.Inputs.xReadyToDry AT %IX."OpcUaDryer".xReadyToDry;
	::gDryerAnc.Inputs.xJamDetection AT %IX."OpcUaDryer".xJamDetection;
	::gDryerAnc.Inputs.xTransportMoving AT %IX."OpcUaDryer".xTransportMoving;
	::gDryerAnc.Inputs.xInRemote AT %IX."OpcUaDryer".xInRemote;
	::gDryerAnc.Parameters.rSpeedSetPoint AT %QD."OpcUaDryer".rBeltSpeedSetPoint;
	::gDryerAnc.Parameters.rMediaLength AT %QD."OpcUaDryer".rBoardLength;
	::gDryerAnc.Parameters.rMediaWidth AT %QD."OpcUaDryer".rBoardWidth;
	::gDryerAnc.Parameters.rMediaThickness AT %QD."OpcUaDryer".rBoardThickness;
	::gDryerAnc.Parameters.rMediaGap AT %QD."OpcUaDryer".rBoardGap;
	::gDryerRemoteData.Signals.xMediaPresent AT %QX."OpcUaDryer".Signals_xMediaPresent;
	::gDryerRemoteData.Signals.xBreakerOKBlowerInput AT %QX."OpcUaDryer".Signals_xBreakerOKBlowerInput;
	::gDryerRemoteData.Signals.xBreakerOKBlowerOutput AT %QX."OpcUaDryer".Signals_xBreakerOKBlowerOutput;
	::gDryerRemoteData.Signals.Safety.xMovementsEnabled AT %QX."OpcUaDryer".Signals_Safety_xMovementsEnabled;
	::gDryerRemoteData.Signals.Safety.xRemoteEStopOK AT %QX."OpcUaDryer".Signals_Safety_xRemoteEStopOK;
	::gDryerRemoteData.Signals.Safety.xEStopFrontOK AT %QX."OpcUaDryer".Signals_Safety_xEStopFrontOK;
	::gDryerRemoteData.Signals.Safety.xEStopRearOK AT %QX."OpcUaDryer".Signals_Safety_xEStopRearOK;
	::gDryerRemoteData.Signals.Safety.xClosedFrontInput AT %QX."OpcUaDryer".Signals_Safety_xClosedFrontIn;
	::gDryerRemoteData.Signals.Safety.xClosedFrontOutput AT %QX."OpcUaDryer".Signals_Safety_xClosedFrontOut;
	::gDryerRemoteData.Signals.Safety.xClosedRearInput AT %QX."OpcUaDryer".Signals_Safety_xClosedRearIn;
	::gDryerRemoteData.Signals.Safety.xClosedRearOutput AT %QX."OpcUaDryer".Signals_Safety_xClosedRearOut;
	::gDryerAnc.Inputs.xError AT %IX."OpcUaDryer".xError;
	::gDryerAnc.Inputs.xInRemote AT %IX."OpcUaDryer".ModuleOk;
END_VAR
```

### Acp10map.ncm - PC_any/Motion/Acp10map.ncm
```
NcMapping (NcSwId=Acp10, DisabledNodesAreHidden=False)
  NcObject gAxis01 (ModuleId=8V1045.00-2_BELT, Type=ncAXIS, Channel=1, AcoposSimulation=Off, InitParameter=BeltP4_i, AcoposParameter=BeltP4_a, Disabled=FALSE, ModuleDisabled=FALSE)
  NcObject 8V1045.00-2_ncV_AXIS1 (ModuleId=8V1045.00-2_BELT, Type=ncV_AXIS, Channel=1, Disabled=TRUE, ModuleDisabled=FALSE)
  NcObject gAxis21 (ModuleId=8V1016.50-2_BK1, Type=ncAXIS, Channel=1, AcoposSimulation=Off, InitParameter=BK1_i, AcoposParameter=BK_sim_a, Disabled=FALSE, ModuleDisabled=FALSE)
  NcObject 8V1016.50-2_ncV_AXIS1 (ModuleId=8V1016.50-2_BK1, Type=ncV_AXIS, Channel=1, Disabled=TRUE, ModuleDisabled=FALSE)
  NcObject gAxis121 (ModuleId=8V1016.50-2_BK2, Type=ncAXIS, Channel=1, AcoposSimulation=Off, InitParameter=BK1_i, AcoposParameter=BK_sim_a, Disabled=FALSE, ModuleDisabled=FALSE)
  NcObject 8V1016.50-2_ncV_AXIS1 (ModuleId=8V1016.50-2_BK2, Type=ncV_AXIS, Channel=1, Disabled=TRUE, ModuleDisabled=FALSE)
  NcObject gAxisStp01 (ModuleId=X67SM2436, ModuleAddress=SDC_IF1.ST1, Type=ncAXIS, Channel=1, AcoposSimulation=Off, InitParameter=SM_i, AcoposParameter=SM_a, Disabled=FALSE, ModuleDisabled=FALSE)
  NcObject gAxisStp02 (ModuleId=X67SM2436, ModuleAddress=SDC_IF1.ST2, Type=ncAXIS, Channel=1, AcoposSimulation=Off, InitParameter=SM_i, AcoposParameter=SM_a, Disabled=FALSE, ModuleDisabled=FALSE)
  NcObject gAxis41 (ModuleId=8V1045.00-2_NCrash1, Type=ncAXIS, Channel=1, AcoposSimulation=Off, InitParameter=NonCrash_i, AcoposParameter=NonCrash_a, Disabled=FALSE, ModuleDisabled=FALSE)
  NcObject 8V1045.00-2_ncV_AXIS1 (ModuleId=8V1045.00-2_NCrash1, Type=ncV_AXIS, Channel=1, Disabled=TRUE, ModuleDisabled=FALSE)
```

## Logical view

Binary libraries used (declarations not repeated): DataObj, operator, runtime, astime, AsCANopen, brsystem, sys_lib, AsSafety, FileIO, standard, AsXml, asstring, AsFifo, AsBrStr, MTTypes, AsTCP, AsIecCon, AsIOAcc, AsBrMath, AsEPL, ArEventLog, AsARCfg, ArProject, AsHttp, dvframe, AsMath, AsSem, AsOpcUas, AsOpcUac, Acp10man 5.21.2, Acp10par 5.21.2, NcGlobal 5.21.2, Acp10sdc 5.21.2, Acp10sim 5.21.2, Acp10_MC 5.21.2, MTBasics 5.16.0, MTFilter 5.16.0, MpAlarmX 5.21.0, MpBase, MpCom, MpServer 5.21.0, AxisFunc, UtMgr 2.01.0, UtWs

### Package Logical/Libraries - Global libraries

### Library Logical/Libraries/BRSE_JSON (ANSIC, version 1.12.0) - Contains FUBs for JSON string handling.
Depends on: sys_lib, astime, AsBrStr

#### BRSE_JSON.typ - Exported data types
```iecst
(********************************************************************
 * COPYRIGHT -- B&R
 ********************************************************************
 * Library: BRSE_JSON
 * File: BRSE_JSON.typ
 * Author: Florian Damerow
 * Created: March 09, 2011
 ********************************************************************
 * Data types of library BRSE_JSON
 ********************************************************************)

TYPE
	TaskDoc1_typ : 	STRUCT
		Output : Output1_typ;
		Input : Input1_typ;
		State : USINT;
	END_STRUCT;
	Input1_typ : 	STRUCT
		StructDepth : DINT;
	END_STRUCT;
	Output1_typ : 	STRUCT
		StatusGet : UINT;
		StatusInfo : UINT;
		StatusSearch : UINT;
	END_STRUCT;
END_TYPE
```

#### BRSE_JSON.var - Exported constants
```iecst
(********************************************************************
 * COPYRIGHT -- B&R
 ********************************************************************
 * Library: BRSE_JSON
 * File: BRSE_JSON.var
 * Author: Florian Damerow
 * Created: April 05, 2011
 ********************************************************************
 * Constants of library BRSE_JSON
 ********************************************************************)
VAR CONSTANT
	MAX_STRUCT_NAME_LENGTH_Parse : UINT := 1000;
	MAX_STRUCT_DEPTH_Stringify : USINT := 20;
	MAX_STRUCT_DEPTH_Parse : USINT := 20;
	MAX_OUTPUT_LENGTH_Stringify : UDINT := 6000;
END_VAR
```

#### example.c
```c
/*! \page Example

\section Example Package
The package contains everything needed to operate an simple JSON server.
By running the included html file in Internet Explorer it is possible to showcase "monitor mode".
To do this the tasks Simulation and GetStruct is necessary. Go to \ref Downloads

*/
```

### Library Logical/Libraries/IecCheck (IEC)

#### IecCheck.st
```iecst
(* Check divisor for SINT division *)
FUNCTION CheckDivSint
	IF divisor=0 THEN
		CheckDivSint:=1;
		MakeEntry(55555,divisor,'CheckDivSint');
	ELSE
		CheckDivSint:=divisor;
	END_IF
END_FUNCTION

(* Check divisor for USINT division *)
FUNCTION CheckDivUsint
	IF divisor=0 THEN
		CheckDivUsint:=1;
		MakeEntry(55555,divisor,'CheckDivUsint');
	ELSE
		CheckDivUsint:=divisor;
	END_IF
END_FUNCTION

(* Check divisor for INT division *)
FUNCTION CheckDivInt
	IF divisor=0 THEN
		CheckDivInt:=1;
		MakeEntry(55555,divisor,'CheckDivInt');
	ELSE
		CheckDivInt:=divisor;
	END_IF
END_FUNCTION

(* Check divisor for UINT division *)
FUNCTION CheckDivUint
	IF divisor=0 THEN
		CheckDivUint:=1;
		MakeEntry(55555,divisor,'CheckDivUint');
	ELSE
		CheckDivUint:=divisor;
	END_IF
END_FUNCTION

(* Check divisor for DINT division *)
FUNCTION CheckDivDint
	IF divisor=0 THEN
		CheckDivDint:=1;
		MakeEntry(55555,divisor,'CheckDivDint');
	ELSE
		CheckDivDint:=divisor;
	END_IF
END_FUNCTION

(* Check divisor for UDINT division *)
FUNCTION CheckDivUdint
	IF divisor=0 THEN
		CheckDivUdint:=1;
		MakeEntry(55555,divisor,'CheckDivUdint');
	ELSE
		CheckDivUdint:=divisor;
	END_IF
END_FUNCTION

(* Check divisor for REAL division *)
FUNCTION CheckDivReal
	IF divisor=0 THEN
		CheckDivReal:=1;
		MakeEntry(55555,0,'CheckDivReal');
	ELSE
		CheckDivReal:=divisor;
	END_IF
END_FUNCTION

(* Check divisor for LREAL division *)
FUNCTION CheckDivLReal
	IF divisor=0 THEN
		CheckDivLReal:=1;
		MakeEntry(55555,0,'CheckDivLReal');
	ELSE
		CheckDivLReal:=divisor;
	END_IF
END_FUNCTION

(* Check range for array access *)
FUNCTION CheckBounds
	IF index < lower THEN
		CheckBounds := lower;
		MakeEntry(55555,index,'CheckBounds');
	ELSIF index > upper THEN
		CheckBounds := upper;
		MakeEntry(55555,index,'CheckBounds');
	ELSE
		CheckBounds := index;
	END_IF
END_FUNCTION

(* Check range for enumeration *)
FUNCTION CheckRange
	IF value < lower THEN
		CheckRange := lower;
		MakeEntry(55555,value,'CheckRange');
	ELSIF value > upper THEN
		CheckRange := upper;
		MakeEntry(55555,value,'CheckRange');
	ELSE
		CheckRange := value;
	END_IF
END_FUNCTION

(* Check range for subrange of signed data types *)
FUNCTION CheckSignedSubrange
	IF value < lower THEN
		CheckSignedSubrange := lower;
		MakeEntry(55555,value,'CheckSignedSubrange');
	ELSIF value > upper THEN
		CheckSignedSubrange := upper;
		MakeEntry(55555,value,'CheckSignedSubrange');
	ELSE
		CheckSignedSubrange := value;
	END_IF
END_FUNCTION

(* Check range for subrange of unsigned data types *)
FUNCTION CheckUnsignedSubrange
	IF value < lower THEN
		CheckUnsignedSubrange := lower;
		MakeEntry(55555,value,'CheckUnsignedSubrange');
	ELSIF value > upper THEN
		CheckUnsignedSubrange := upper;
		MakeEntry(55555,value,'CheckUnsignedSubrange');
	ELSE
		CheckUnsignedSubrange := value;
	END_IF
END_FUNCTION

(* Check address when reading dynamic variables *)
FUNCTION CheckReadAccess
	IF address=0 THEN
		(* TODO: Insert an appropriate code, see AutomationStudio help for further information *)
		MakeEntry(55555,address,'Read from NULL');
	END_IF

	CheckReadAccess:=0;
END_FUNCTION

(* Check address when writing dynamic variables *)
FUNCTION CheckWriteAccess
	IF address=0 THEN
		(* TODO: Insert an appropriate code, see AutomationStudio help for further information *)
		MakeEntry(55555,address,'Write to NULL');
	END_IF

	CheckWriteAccess:=0;
END_FUNCTION

(* Makes an entry (log book entry) in the error log book *)
FUNCTION MakeEntry
	status_name := ST_name(0,ADR(taskname),ADR(group));

	brsstrcpy(ADR(out_text),ADR(text));
	brsstrcat(ADR(out_text),ADR(' > in task > '));
	brsstrcat(ADR(out_text),ADR(taskname));
	brsitoa(USINT_TO_DINT(group),ADR(aux_text));
	brsstrcat(ADR(out_text),ADR('. Group: '));
	brsstrcat(ADR(out_text),ADR(aux_text));
	brsitoa(index,ADR(aux_text));
	brsstrcat(ADR(out_text),ADR('. Index: '));
	brsstrcat(ADR(out_text),ADR(aux_text));

	MakeEntry := ADR(out_text);
	ERRxfatal(number,index,ADR(out_text));

END_FUNCTION
```

### Library Logical/Libraries/ErrACS380 (IEC)

#### Constants.var - Exported constants
```iecst
VAR CONSTANT
	MAX_ERR_LIST : UINT := 199;
END_VAR
```

#### ErrMessage.st
```iecst
(*<$Description$> Takes the error list and the current error ID and gives back the message associated </$Description$>*)
FUNCTION_BLOCK ErrMessage

	CASE Internal.Step OF
		// -----------------------------------------------------------------
		0: 		(* DISABLED *)

			Status	:= DISABLED;

			IF Enable THEN
				Internal.Step	:= 1;
			END_IF

		// -----------------------------------------------------------------
		1:		(* WAITING *)

			Status	:= STATUS_OK;

			IF NewID THEN
				NewID			:= FALSE;
				Internal.Step	:= 2;
			END_IF

		// -----------------------------------------------------------------
		2: 		(* BUSY *)

			Status	:= ACS380_BUSY;

			FOR Internal.Counter := 0 TO MAX_ERR_LIST DO

				IF ErrList[Internal.Counter].ErrorID = CurrentErrID THEN

					CurrentErrMessage		:= ErrList[Internal.Counter].ErrorText;
					Internal.ErrNotFound	:= FALSE;
					Internal.Step			:= 3;
					EXIT;

				ELSE

					Internal.ErrNotFound	:= TRUE;

				END_IF

			END_FOR

			IF Internal.ErrNotFound THEN
				Internal.StatusError	:= TRUE;
				Internal.Step			:= 9;
			END_IF

		// -----------------------------------------------------------------
		3:		(* DONE *)

			Status	:= DONE;

			IF NewID THEN
				NewID			:= FALSE;
				Internal.Step	:= 2;
			END_IF

		// -----------------------------------------------------------------
		9:	(* ERROR *)

			Status	:= ERR;

			IF NewID THEN
				NewID			:= FALSE;
				Internal.Step	:= 2;
			END_IF

	END_CASE

END_FUNCTION_BLOCK
```

### Package Logical/ExtPack - External Packages

### Program Logical/ExtPack/_Ancillaries/DryerCtrl/DryerCtrl_v1/DryerCtrl (IEC)

#### DryerCtrl.var
```iecst
VAR
	Dryer : REFERENCE TO DryerAnc_typ;
	AlarmsReseted : DryerAlarms_typ;
	CommandsReseted : DryerCommands_typ;
	tiTimeToEmpty : TIME;
	tonEmptyBelt : TON;
	xStartTransportAndPrepare : BOOL;
	OutputsReset : DryerOutputs_typ;
	iDryerModel : USINT;
	iIndexHistory : USINT;
	StateHistory : ARRAY[0..iHistoryLines] OF DryerCtrlStatus_enum;
END_VAR
VAR CONSTANT
	iHistoryLines : USINT := 20;
END_VAR
```

#### Configuration.st
```iecst
ACTION Configuration:

	CASE Dryer.Status.DryerType OF
		DRYERTY_EFI:
			Dryer.Parameters.Hw.iMaxMediaWidth := 1800;
			Dryer.Parameters.Hw.iMaxMediaLength := 3000;
			Dryer.Parameters.Hw.rDryerLength := 5000.0;
			Dryer.Parameters.Hw.xDoubleLineAllowed := TRUE;

	END_CASE

END_ACTION
```

#### Dryer.st
```iecst
PROGRAM _CYCLIC

	Dryer ACCESS ADR(gDryerAnc);

//	Dryer.Status.Version.iVersion0 := ;
//	Dryer.Status.Version.iVersion1 := ;
//	Dryer.Status.Version.iVersion2 := ;
//	Dryer.Status.Version.iVersion3 := ;

	//Model evaluation
	iDryerModel.0 := Dryer.Inputs.xModelInput[0];
	iDryerModel.1 := Dryer.Inputs.xModelInput[1];
	iDryerModel.2 := Dryer.Inputs.xModelInput[2];

	Dryer.Parameters.xInstalled := iDryerModel>0;

	//Specify Type of primer Model
	Dryer.Status.iModel := iDryerModel;
	CASE iDryerModel OF
		1: Dryer.Status.DryerType := DRYERTY_EFI;
		ELSE Dryer.Status.DryerType := DRYERTY_UNDEFINED;
	END_CASE

	IF NOT Dryer.Parameters.xInstalled OR NOT Dryer.ParSw.xEnabled THEN
		ResetAlarms;
		Dryer.Outputs := OutputsReset;
		Dryer.Commands:=CommandsReseted;
		Dryer.Status.DeviceStatus:= DRYER_TURNED_OFF;
		UpdateStatus;
		RETURN;
	END_IF

	IF Dryer.Commands.xResetAlarms THEN ResetAlarms; END_IF

	Configuration;

	Status;

	Alarms;

	IF Dryer.Status.Device.xFaulted OR Dryer.Status.Device.xTurnedOff OR NOT Dryer.Parameters.xLineInAuto THEN
		Dryer.Status.CtrlStatus:=DRYERCTRL_STOPPED;
	END_IF

	CASE Dryer.Status.CtrlStatus OF
		DRYERCTRL_STOPPED:
			Dryer.Outputs := OutputsReset;

			IF Dryer.Status.DeviceStatus=DRYER_INIT AND (Dryer.Commands.xStartTransport OR Dryer.Commands.xPrepare) THEN
				IF Dryer.Commands.xPrepare THEN
					xStartTransportAndPrepare := TRUE;
				END_IF
				Dryer.Status.CtrlStatus:=DRYERCTRL_PREPARINGTOMOVE;
			END_IF

			IF  Dryer.Status.DeviceStatus=DRYER_INIT AND Dryer.Commands.xBelEmpty THEN
				Dryer.Status.CtrlStatus := DRYERCTRL_PREPARINGEMPTYBELT;
			END_IF

		DRYERCTRL_PREPARINGEMPTYBELT:
			Dryer.Outputs.xPrepareToEmptyBelt := TRUE;
			IF Dryer.Inputs.xReadyToEmptyBelt THEN
				Dryer.Status.CtrlStatus := DRYERCTRL_PREPARINGTOMOVE;
			END_IF

		DRYERCTRL_STOPPING:
			//Actions
			Dryer.Outputs := OutputsReset;

			//Transition
			IF Dryer.Status.DeviceStatus=DRYER_TURNED_OFF OR Dryer.Status.DeviceStatus=DRYER_INIT THEN
				Dryer.Status.CtrlStatus:=DRYERCTRL_STOPPED;
			END_IF

		DRYERCTRL_CONTROLSTOPPING:
			//Wait to have the belt empty and send the Stop order
			IF Dryer.Status.xBeltEmpty OR NOT Dryer.Inputs.xTransportMoving THEN
				Dryer.Status.CtrlStatus:=DRYERCTRL_STOPPING;
			END_IF

		DRYERCTRL_PREPARINGTOMOVE:
			Dryer.Outputs.xPrepareToEmptyBelt := FALSE;
			Dryer.Outputs.xRunTransport:=TRUE;
			IF Dryer.Status.DeviceStatus=DRYER_BELTRUNNING THEN
				Dryer.Status.CtrlStatus:=DRYERCTRL_MOVING;
			END_IF

		DRYERCTRL_MOVING:
			IF Dryer.Commands.xPrepare OR xStartTransportAndPrepare THEN
				xStartTransportAndPrepare := FALSE;
				Dryer.Status.CtrlStatus:=DRYERCTRL_PREPARING;
			END_IF

		DRYERCTRL_PREPARING:
			Dryer.Outputs.xPrepareToDry:=TRUE;
			IF Dryer.Status.DeviceStatus=DRYER_READY THEN
				Dryer.Status.CtrlStatus:=DRYERCTRL_PREPARED;
			END_IF

		DRYERCTRL_PAUSED,
		DRYERCTRL_PREPARED:
			IF Dryer.Commands.xStart THEN
				Dryer.Status.CtrlStatus:=DRYERCTRL_STARTING;
			END_IF

		DRYERCTRL_STARTING:
			//Actions
			Dryer.Outputs.xStartDrying:=TRUE;
			//Transition
			IF Dryer.Status.DeviceStatus=DRYER_DRYING THEN
				Dryer.Status.CtrlStatus:=DRYERCTRL_DRYING;
			END_IF
			//Transition
			IF Dryer.Commands.xPause THEN
				Dryer.Status.CtrlStatus:=DRYERCTRL_PAUSING;
			END_IF

		DRYERCTRL_DRYING:
			IF Dryer.Commands.xPause THEN
				Dryer.Status.CtrlStatus:=DRYERCTRL_PAUSING;
			END_IF

		DRYERCTRL_PAUSING:
			//Wait to empty the Belt to avoid media inside
			IF Dryer.Status.xBeltEmpty THEN
				Dryer.Outputs.xStartDrying:=FALSE;
				//Transition
				IF Dryer.Status.DeviceStatus=DRYER_READY THEN
					Dryer.Status.CtrlStatus:=DRYERCTRL_PAUSED;
				END_IF
			END_IF

			IF Dryer.Commands.xStart THEN
				Dryer.Status.CtrlStatus:=DRYERCTRL_STARTING;
			END_IF

	END_CASE

	IF Dryer.Commands.xStop THEN
		Dryer.Status.CtrlStatus:=DRYERCTRL_STOPPING;
	ELSIF Dryer.Commands.xControlStop THEN
		Dryer.Status.CtrlStatus:=DRYERCTRL_CONTROLSTOPPING;
	END_IF

	//Store the history of the status to easy the debug
	IF Dryer.Status.CtrlStatus<>StateHistory[0] THEN
		FOR iIndexHistory:=iHistoryLines TO 1 BY -1 DO
			StateHistory[iIndexHistory]:=StateHistory[iIndexHistory-1];
		END_FOR;
		StateHistory[0]:=Dryer.Status.CtrlStatus;
	END_IF

	//Reset all commands
	Dryer.Commands:=CommandsReseted;

END_PROGRAM
```

### Dryer.typ
```iecst
TYPE
	DryerCtrlStatus_enum :
		(
		DRYERCTRL_STOPPED,
		DRYERCTRL_STOPPING,
		DRYERCTRL_PREPARING,
		DRYERCTRL_PREPARED,
		DRYERCTRL_PAUSING,
		DRYERCTRL_PAUSED,
		DRYERCTRL_STARTING,
		DRYERCTRL_DRYING,
		DRYERCTRL_CONTROLSTOPPING,
		DRYERCTRL_PREPARINGTOMOVE,
		DRYERCTRL_MOVING,
		DRYERCTRL_PREPARINGEMPTYBELT
		);
	DryerStatus_enum :
		(
		DRYER_TURNED_OFF,
		DRYER_INIT,
		DRYER_PREPARING,
		DRYER_READY,
		DRYER_DRYING,
		DRYER_FAULTED,
		DRYER_DRYING_ARC_LAMP,
		DRYER_BELTRUNNING
		);
	DryerType_enum :
		(
		DRYERTY_UNDEFINED,
		DRYERTY_EFI (*EFI manufacturer.*)
		);
	DryerInputs_typ : 	STRUCT
		xError : BOOL;
		xDrying : BOOL;
		xReadyToDry : BOOL;
		xJamDetection : BOOL;
		xTransportMoving : BOOL;
		xInRemote : BOOL;
		xModelInput : ARRAY[0..2]OF BOOL;
		xMediaPresent : BOOL;
		xCommsOK : BOOL; (*Modbus communications are working properly*)
		xBeltEmpty : BOOL; (*Belt empty in the device*)
		xReadyToEmptyBelt : BOOL; (*Dryer ready to perform empty belt*)
		xStopButtonPressed : BOOL; (*Red button pressed. Stop Required*)
	END_STRUCT;
	DryerOutputs_typ : 	STRUCT
		xPrepareToDry : BOOL;
		xStartDrying : BOOL;
		xRunTransport : BOOL;
		xPrepareToEmptyBelt : BOOL;
	END_STRUCT;
	DryerAlarms_typ : 	STRUCT
		xError : BOOL;
		xStopRequest : BOOL; (*Stop request from Dryer when physical stop button is pressed*)
		xNotRemote : BOOL;
		xNoDryerPresent : BOOL;
		xAnyAlarm : BOOL;
		xCriticalAlarm : BOOL;
		xWarningAlarm : BOOL;
		xCommsError : BOOL;
	END_STRUCT;
	DryerParametersHw_typ : 	STRUCT
		iMaxMediaWidth : UINT; (*Maximum media width allowed in mm*)
		iMinMediaWidth : UINT; (*Minimum media width allowed in mm*)
		iMaxMediaLength : UINT; (*Maximum media length allowed in mm*)
		iMinMediaLength : UINT; (*Minimum media length allowed in mm*)
		rDryerLength : REAL; (*Length in mm*)
		rMaxSpeed : REAL := 100.0; (*Maximum speed allowed in m/min*)
		xDoubleLineAllowed : BOOL; (*Active when printer allows double line printing*)
	END_STRUCT;
	DryerParametersSw_typ : 	STRUCT
		xEnabled : BOOL;
		xEnableNIR : BOOL;
		xEnableDDC : BOOL; (*Enable DDC behavior in Dryer*)
		xEnableArcLamp : BOOL;
		rSubstratePowerReduction : REAL := 1.0; (*Substrate power reduction. From 1.0 (default) to 0.3 is allowed*)
	END_STRUCT;
	DryerParameters_typ : 	STRUCT
		xInstalled : BOOL;
		xSimulationMode : BOOL; (*Defined by the configuration in Automation Studio*)
		xCommsOK : BOOL;
		xAlrPresent : BOOL;
		LineState : LineStatus_enum;
		xLineInAuto : BOOL;
		xInRemote : BOOL;
		xSecurityOK : BOOL;
		rSpeedSetPoint : REAL; (*Speed in m/min*)
		rMediaLength : REAL; (*Length in mm*)
		rMediaWidth : REAL; (*Length in mm*)
		rMediaThickness : REAL; (*Length in mm*)
		rMediaGap : REAL; (*Length in mm*)
		xPreviousDeviceStopped : BOOL;
		LineStatusSummary : LineControlStatusSummarized;
		rDocumentWidth : REAL; (*Length in mm*)
		rDocumentLength : REAL; (*Length in mm*)
		rDocumentOffsetL1 : REAL; (*Job's document offset L1 in mm*)
		rDocumentOffsetL2 : REAL; (*Job's document offset L2 in mm*)
		Hw : DryerParametersHw_typ;
		xDoubleLine : BOOL;
	END_STRUCT;
	DryerCommands_typ : 	STRUCT
		xBelEmpty : BOOL; (*Edge commands. Reseted when managed*)
		xStart : BOOL; (*Edge commands. Reseted when managed*)
		xPrepare : BOOL; (*Edge commands. Reseted when managed*)
		xPause : BOOL; (*Edge commands. Reseted when managed*)
		xStop : BOOL; (*Edge commands. Reseted when managed*)
		xControlStop : BOOL; (*Edge commands. Reseted when managed*)
		xStartTransport : BOOL; (*Edge commands. Reseted when managed*)
		xThereIsDryer : BOOL;
		xResetAlarms : BOOL;
	END_STRUCT;
	DryerDeviceStatus_typ : 	STRUCT
		xTurnedOff : BOOL;
		xInit : BOOL;
		xPreparing : BOOL;
		xBeltRunning : BOOL;
		xReadyToDry : BOOL;
		xDrying : BOOL;
		xFaulted : BOOL;
	END_STRUCT;
	DryerStatus_typ : 	STRUCT
		iModel : USINT := 1; (*Model of the Device. 0:BDT 1:Serra*)
		Version : EFI_version_typ;
		CtrlStatus : DryerCtrlStatus_enum;
		DeviceStatus : DryerStatus_enum;
		Device : DryerDeviceStatus_typ;
		xBeltEmpty : BOOL;
		DryerType : DryerType_enum;
	END_STRUCT;
	DryerAnc_typ : 	STRUCT
		Inputs : DryerInputs_typ;
		Outputs : DryerOutputs_typ;
		Alarms : DryerAlarms_typ;
		ParSw : DryerParametersSw_typ;
		Parameters : DryerParameters_typ;
		Commands : DryerCommands_typ;
		Status : DryerStatus_typ;
	END_STRUCT;
END_TYPE
```

### Program Logical/ExtPack/_Ancillaries/FeederCtrl/FeederCtrl_v1/FeederCtrl (IEC)

#### AssignDataComms.st
```iecst
ACTION AssignDataComms:

	//Active modbus slave diagnosis when ancillary is enabled. This parameter must remain to TRUE from then on.
	//Just would be set to FALSE via UaExpert, to reset historic errors when ancillary is disabled
	Feeder.Parameters.xActiveSlaveDiagnosis := TRUE;

	FOR iIndexMedia:=1 TO 4 DO
		iMedia := iMedia + gToWriteDataModbFeeder[iIndexMedia];
	END_FOR

	IF iPreviousMedia <> iMedia THEN
		xNewMediaParameters := TRUE;
		iPreviousMedia := iMedia;
	ELSIF ton_NexMediaParamaters.Q THEN
		xNewMediaParameters := FALSE;
	END_IF

	ton_NexMediaParamaters(IN:=xNewMediaParameters, PT:=T#200MS);

	/////////////////
	//Pre bits treatment
	Feeder.Outputs.Comms.iControl.0 := Feeder.ParSw.xBatchFeeding;
	Feeder.Outputs.Comms.iControl.1 := xNewMediaParameters;
	//Feeder.Outputs.Comms.iControl.2 := ;
	Feeder.Outputs.Comms.iControl.3 := Feeder.Commands.xNewOrder;
	Feeder.Outputs.Comms.iControl.4 := Feeder.Commands.xResetAlarms;
	Feeder.Outputs.Comms.iControl.5 := Feeder.Commands.xSheetFeeding;
	Feeder.Outputs.Comms.iControl.6 := Feeder.Commands.xStopFeeding;

	//Write Registers
	gToWriteDataModbFeeder[1] := REAL_TO_UINT(Feeder.Parameters.Media.rLength*10);
	gToWriteDataModbFeeder[2] := REAL_TO_UINT(Feeder.Parameters.Media.rWidth*10);
	gToWriteDataModbFeeder[3] := REAL_TO_UINT(Feeder.Parameters.Media.rThickness*10);
	gToWriteDataModbFeeder[4] := REAL_TO_UINT(Feeder.Parameters.Media.rGap*10);
	//gToWriteDataModbFeeder[5] := ;
	gToWriteDataModbFeeder[6] := Feeder.Parameters.iLineConfig;
	gToWriteDataModbFeeder[7] := Feeder.Parameters.iRegisterType;
	gToWriteDataModbFeeder[8] := REAL_TO_UINT(Feeder.Parameters.Media.rOffsetRegisterL1);
	gToWriteDataModbFeeder[9] := Feeder.Outputs.Comms.iControl;
	gToWriteDataModbFeeder[10] := REAL_TO_UINT(Feeder.Parameters.Media.rOffsetRegisterL2);
	gToWriteDataModbFeeder[11] := REAL_TO_UINT(Feeder.Parameters.rBeltSpeedSetPoint*10);
	//gToWriteDataModbFeeder[12] := ;
	gToWriteDataModbFeeder[13] := Feeder.Parameters.iCentralOffset;
	gToWriteDataModbFeeder[14] := Feeder.Parameters.iCounterSetPointL1;
	gToWriteDataModbFeeder[15] := Feeder.Parameters.iCounterSetPointL2;
	(*
	gToWriteDataModbFeeder[16] := ;
	gToWriteDataModbFeeder[17] := ;
	gToWriteDataModbFeeder[18] := ;
	gToWriteDataModbFeeder[19] := ;
	gToWriteDataModbFeeder[20] := ;
	gToWriteDataModbFeeder[21] := ;
	gToWriteDataModbFeeder[22] := ;
	gToWriteDataModbFeeder[23] := ;
	gToWriteDataModbFeeder[24] := ;
	gToWriteDataModbFeeder[25] := ;
	*)

	//Disabling writting after some time active. To test
	tonDisableWrittingOfData.IN:= NOT xDisableWriteData;
	tonDisableWrittingOfData.PT:= T#1000ms;
	tonDisableWrittingOfData();

	IF tonDisableWrittingOfData.Q THEN
		xDisableWriteData := TRUE;
	END_IF

	FOR iIndex:=1 TO 25 DO
		IF gToWriteDataModbFeeder[iIndex]<>CopyOfWriteData[iIndex] THEN
			xDisableWriteData := FALSE;
		END_IF
	END_FOR

	Feeder.Orders.xDisableWriteBlock := xDisableWriteData;

	//Copying previous data
	CopyOfWriteData := gToWriteDataModbFeeder;

	////////////////
	//Read Registers
	IF Feeder.Status.Comms.xModuleOk THEN
		Feeder.Inputs.Comms.iNumBoardsRemainingL1 := gReceivedDataModbFeeder[1];
		Feeder.Inputs.Comms.iNumBoardsRemainingL2 := gReceivedDataModbFeeder[2];
		Feeder.Inputs.Comms.iAlarmWord1 := gReceivedDataModbFeeder[3];
		Feeder.Inputs.Comms.iAlarmWord2 := gReceivedDataModbFeeder[4];
		Feeder.Inputs.Comms.iAlarmWord3 := gReceivedDataModbFeeder[5];
		Feeder.Inputs.Comms.iAlarmWord4 := gReceivedDataModbFeeder[6];
		Feeder.Inputs.Comms.iAlarmWord5 := gReceivedDataModbFeeder[7];
		Feeder.Inputs.Comms.iAlarmWord6 := gReceivedDataModbFeeder[8];
		Feeder.Inputs.Comms.iStatus := gReceivedDataModbFeeder[9];
		Feeder.Inputs.Comms.iAlarmWord7 := gReceivedDataModbFeeder[10];
		Feeder.Inputs.Comms.iAlarmWord8 := gReceivedDataModbFeeder[11];
		Feeder.Inputs.Comms.iAlarmWord9 := gReceivedDataModbFeeder[12];
		Feeder.Inputs.Comms.iAlarmWord10 := gReceivedDataModbFeeder[13];
		Feeder.Inputs.Comms.iAlarmWord11 := gReceivedDataModbFeeder[14];
		Feeder.Inputs.Comms.iAlarmWord12 := gReceivedDataModbFeeder[15];
		Feeder.Inputs.Comms.iNumFedBoards := gReceivedDataModbFeeder[16];
		Feeder.Inputs.Comms.iAlarmWord13 := gReceivedDataModbFeeder[17];
		Feeder.Inputs.Comms.iAlarmWord14 := gReceivedDataModbFeeder[18];
		Feeder.Inputs.Comms.iAlarmWord15 := gReceivedDataModbFeeder[19];
		Feeder.Inputs.Comms.iVersion1 := gReceivedDataModbFeeder[20];
		Feeder.Inputs.Comms.iVersion2 := gReceivedDataModbFeeder[21];
		Feeder.Inputs.Comms.iVersion3 := gReceivedDataModbFeeder[22];
		Feeder.Inputs.Comms.iVersion4 := gReceivedDataModbFeeder[23];
		//:= gReceivedDataModbFeeder[24];
		//:= gReceivedDataModbFeeder[25];
	END_IF

	//Post bit treatment
	Feeder.Inputs.Comms.xRemote := Feeder.Inputs.Comms.iStatus.0;
	Feeder.Inputs.Comms.xAlarmPresent := Feeder.Inputs.Comms.iStatus.1;
	Feeder.Inputs.Comms.xPositionReady := Feeder.Inputs.Comms.iStatus.2;
	Feeder.Inputs.Comms.xOrderEnd := Feeder.Inputs.Comms.iStatus.3;
	Feeder.Inputs.Comms.xMinimumStackLevelL1 := Feeder.Inputs.Comms.iStatus.4;
	Feeder.Inputs.Comms.xMinimumStackLevelL2 := Feeder.Inputs.Comms.iStatus.5;
	Feeder.Inputs.Comms.xEnableFeeding := Feeder.Inputs.Comms.iStatus.6;
	Feeder.Inputs.Comms.xOnline := Feeder.Inputs.Comms.iStatus.7;

END_ACTION
```

#### FeederCtrl.var - Local variables
```iecst
VAR
	Feeder : REFERENCE TO Feeder_typ;
	AlarmsReseted : FeederAlarms_typ;
	ResetCommands : FeederCommands_typ;
	tonNotOnline : TON;
	CommsReset : FeederCommsInputs_typ;
	OutputsReset : FeederOutputs_typ;
	PhysicalOutputsReset : FeederPhysicalOutputs_typ;
	iMedia : UINT;
	iPreviousMedia : UINT;
	ton_NexMediaParamaters : TON;
	xNewMediaParameters : BOOL;
	iIndexMedia : UINT;
	iFeederModel : USINT;
	iIndexHistory : USINT;
	StateHistory : ARRAY[0..iHistoryLines] OF FeederCtrlStatus_enum;
END_VAR
VAR CONSTANT
	iHistoryLines : USINT := 20;
END_VAR
VAR
	ModSlaveState : UINT;
	LastError : UINT;
	LastErrorBlockNum : UINT;
	CopyOfWriteData : ARRAY[1..25] OF UINT;
	tonDisableWrittingOfData : TON;
	xDisableWriteData : BOOL;
	ton_CommsError : TON;
	EraseWriteData : ARRAY[1..25] OF UINT;
END_VAR
```

### Program Logical/ExtPack/_Ancillaries/FeederCtrl/FeederSim/FeederSim_v1/FeederSim (IEC)

#### FeederSim.st - Init, cyclic, exit code
```iecst
PROGRAM _INIT

	Feeder ACCESS ADR(gFeeder);
	SimFeeder ACCESS ADR(gSimFeeder);

	Feeder.Status.Comms.xModuleOk := TRUE;

END_PROGRAM

PROGRAM _CYCLIC
	(* Insert code here *)
	Feeder ACCESS ADR(gFeeder);
	SimFeeder ACCESS ADR(gSimFeeder);

	Feeder.Inputs.xFeederPresent:=TRUE;
	Feeder.Inputs.xOnline:=TRUE;
	Feeder.Inputs.Comms.xRemote := TRUE;
	Feeder.Inputs.xError:=SimFeeder.Commands.CreateError;

	tonPrepare.IN:=	Feeder.Outputs.Physical.xPrepareToFeed;
	tonPrepare.PT:= T#2s;
	tonPrepare();
	Feeder.Inputs.xReadyToFeed:=tonPrepare.Q;

	tonFeed.IN:= Feeder.Inputs.xReadyToFeed AND Feeder.Outputs.Physical.xStartFeeding;
	tonFeed.PT:= T#1s;
	tonFeed();
	Feeder.Inputs.xFeeding:=tonFeed.Q;

	Feeder.Inputs.Comms.iVersion1 := 1;
	Feeder.Inputs.Comms.iVersion2 := 1;
	Feeder.Inputs.Comms.iVersion3 := 3;
	Feeder.Inputs.Comms.iVersion4 := 15;

END_PROGRAM
```

#### FeederSim.var - Local variables
```iecst
VAR
	SimFeeder : REFERENCE TO FeederSim_typ;
	Feeder : REFERENCE TO Feeder_typ;
	tonPrepare : TON;
	tonFeed : TON;
END_VAR
```

### Program Logical/ExtPack/_Ancillaries/OpvCtrl/OpvCtrl_v1/OpvCtrl

#### OpvCtrl.var
```iecst
VAR
	OverVarnish : REFERENCE TO Opv_typ;
	AlarmsReseted : OPVAlarms_typ;
	ResetCommands : OPVCommands_typ;
	xEnablePriming : BOOL; (*Active if priming is enabled from SW and from Printer/Line*)
	tiTimeToEmpty : TIME;
	tonEmptyBelt : TON;
	CommsReset : OPVCommsInputs_typ;
	OutputsReset : OPVOutputs_typ;
	PhysicalOutputsReset : OPVPhysicalOutputs_typ;
	iOpvModel : USINT;
	iIndexHistory : USINT;
	StateHistory : ARRAY[0..iHistoryLines] OF OPVCtrlStatus_enum;
END_VAR
VAR CONSTANT
	iHistoryLines : USINT := 20;
END_VAR
VAR
	rPrevWidth : REAL;
	rPrevGap : REAL;
	rPrevThickness : REAL;
	rPrevLength : REAL;
	xBoardParametersChanged : BOOL;
	tof_BoardParametersChanged : TOF;
	ModSlaveState : UINT;
	LastError : UINT;
	LastErrorBlockNum : UINT;
	CopyOfWriteData : ARRAY[1..25] OF UINT;
	tonDisableWrittingOfData : TON;
	xDisableWriteData : BOOL;
	ton_CommsError : TON;
	EraseWriteData : ARRAY[1..25] OF UINT;
END_VAR
```

#### Alarms.st
```iecst
ACTION Alarms:

	OverVarnish.Alarms.xNoOPVPresent:= NOT OverVarnish.Inputs.xOPVPresent;

	//IF NO OverVarnish, define that alarm and exit
	IF OverVarnish.Alarms.xNoOPVPresent THEN
		ResetAlarms;
		OverVarnish.Alarms.xNoOPVPresent:=TRUE;
	END_IF

	//OverVarnish No Powered Warning
	IF OverVarnish.Inputs.xNoPowered THEN OverVarnish.Alarms.xNoPowered := TRUE; END_IF

	OverVarnish.Alarms.xCoatingLevelLow:=OverVarnish.Inputs.xCoatingLevelLow;

	IF OverVarnish.Inputs.xError THEN
		OverVarnish.Alarms.xError := TRUE;
	END_IF

	//Saving modbus slave status when comms error raises
	IF EDGEPOS (OverVarnish.Alarms.xCommsError) THEN
		ModSlaveState := OverVarnish.Status.Comms.ModSlaveState;
		LastError := OverVarnish.Status.Comms.LastError;
		LastErrorBlockNum := OverVarnish.Status.Comms.LastErrorBlockNum;
	END_IF

	//Alarms related to comms
	IF OverVarnish.Status.Comms.xModuleOk THEN
		//Remote
		IF (NOT OverVarnish.Inputs.Comms.xRemote) AND OverVarnish.Parameters.xLineInAuto THEN
			OverVarnish.Alarms.xNotRemote := TRUE;
		END_IF

		//Stop request
		IF OverVarnish.Inputs.Comms.xStopButtonPressed THEN
			OverVarnish.Alarms.xStopRequest := TRUE;
		END_IF
	END_IF

	//Data write to ancillaries is critical to be updated properly. So just write block is monitored to raise comms alarm
	//Added ancillary first command used to get it ready to check comms also.
	//Read function not considered as the only variable critical for line process is to acknowledge "belt empty" status and in case of module nOk
	//timer "tonEmptyBelt" is executed
	ton_CommsError.IN := NOT OverVarnish.Status.Comms.xModuleOk AND (NOT OverVarnish.Orders.xDisableWriteBlock OR OverVarnish.Commands.xPrepare);
	ton_CommsError.PT := T#500ms;
	ton_CommsError();

	IF ton_CommsError.Q  THEN
		OverVarnish.Alarms.xCommsError := TRUE;
	END_IF

	//Alarms Summary
	//Critical
	OverVarnish.Alarms.xCriticalAlarm:= OverVarnish.Alarms.xError OR
										OverVarnish.Alarms.xNoPowered OR
										OverVarnish.Alarms.xNotRemote OR
										OverVarnish.Alarms.xStopRequest OR
										OverVarnish.Alarms.xCommsError;

	//Warning
	//OverVarnish.Alarms.xWarningAlarm	:=	;

END_ACTION

ACTION ResetAlarms:
	OverVarnish.Alarms := AlarmsReseted;
END_ACTION
```

#### Configuration.st
```iecst
ACTION Configuration:

	CASE OverVarnish.Status.OpvType OF
		OPVTY_GIARDINA:
			OverVarnish.Parameters.Hw.iMaxMediaWidth := 1800;
			OverVarnish.Parameters.Hw.iMaxMediaLength := 3000;
			OverVarnish.Parameters.Hw.rOPVLength := 3000;
			OverVarnish.Parameters.Hw.iMinMediaThickness := 8;
			OverVarnish.Parameters.Hw.iMaxMediaThickness := 160;
			OverVarnish.Parameters.Hw.xDoubleLineAllowed := TRUE;

		OPVTY_DMS:
			OverVarnish.Parameters.Hw.iMaxMediaWidth := 1800;
			OverVarnish.Parameters.Hw.iMaxMediaLength := 3000;
			OverVarnish.Parameters.Hw.rOPVLength := 3000;
			OverVarnish.Parameters.Hw.iMinMediaThickness := 1;
			OverVarnish.Parameters.Hw.iMaxMediaThickness := 150;
			OverVarnish.Parameters.Hw.xDoubleLineAllowed := TRUE;

		OPVTY_TECLIGHTING:
			OverVarnish.Parameters.Hw.iMaxMediaWidth := 1800;
			OverVarnish.Parameters.Hw.iMaxMediaLength := 3200;
			OverVarnish.Parameters.Hw.rOPVLength := 2500;
			OverVarnish.Parameters.Hw.iMinMediaThickness := 3;
			OverVarnish.Parameters.Hw.iMaxMediaThickness := 120;
			OverVarnish.Parameters.Hw.xDoubleLineAllowed := FALSE;

	END_CASE

END_ACTION
```

#### Status.st
```iecst
ACTION Status:

	CASE OverVarnish.Status.DeviceStatus OF
		OPV_TURNED_OFF:
			IF OverVarnish.Inputs.xOPVPresent THEN
				OverVarnish.Status.DeviceStatus:=OPV_INIT;
			END_IF

		OPV_INIT:
			IF NOT OverVarnish.Inputs.xOPVPresent THEN
				OverVarnish.Status.DeviceStatus:=OPV_TURNED_OFF;
			ELSIF OverVarnish.Outputs.Physical.xPrepareToPrime OR OverVarnish.Outputs.Physical.xRunTransport THEN
				OverVarnish.Status.DeviceStatus:=OPV_PREPARING;
			END_IF

		OPV_PREPARING:
			IF OverVarnish.Inputs.xTransportMoving THEN
				OverVarnish.Status.DeviceStatus:=OPV_BELT_RUNNING;
			ELSIF NOT OverVarnish.Outputs.Physical.xPrepareToPrime AND NOT OverVarnish.Outputs.Physical.xRunTransport THEN
				OverVarnish.Status.DeviceStatus:=OPV_INIT;
			END_IF

		OPV_BELT_RUNNING:
			IF NOT OverVarnish.Inputs.xTransportMoving THEN
				OverVarnish.Status.DeviceStatus:=OPV_INIT;
			END_IF
			IF OverVarnish.Inputs.xReadyToPrime THEN
				OverVarnish.Status.DeviceStatus:=OPV_READY;
			END_IF

		OPV_READY:
			IF NOT OverVarnish.Inputs.xReadyToPrime THEN
				OverVarnish.Status.DeviceStatus:=OPV_BELT_RUNNING;
			END_IF
			IF OverVarnish.Inputs.xCoating THEN
				OverVarnish.Status.DeviceStatus:=OPV_PRIMING;
			END_IF

		OPV_PRIMING:
			IF NOT OverVarnish.Inputs.xCoating THEN
				OverVarnish.Status.DeviceStatus:=OPV_READY;
			END_IF
			IF OverVarnish.Inputs.xDryerInRun THEN
				OverVarnish.Status.DeviceStatus:=OPV_DRYING;
			END_IF

		OPV_DRYING:
			IF NOT OverVarnish.Inputs.xDryerInRun THEN
				OverVarnish.Status.DeviceStatus:=OPV_PRIMING;
			END_IF

		OPV_FAULTED:
			IF NOT OverVarnish.Inputs.xError THEN
				OverVarnish.Status.DeviceStatus:=OPV_TURNED_OFF;
			END_IF

	END_CASE

	IF NOT OverVarnish.Inputs.xOPVPresent THEN
		OverVarnish.Status.DeviceStatus:=OPV_TURNED_OFF;
	END_IF
	IF OverVarnish.Status.DeviceStatus <> OPV_TURNED_OFF AND OverVarnish.Inputs.xError THEN
		OverVarnish.Status.DeviceStatus:=OPV_FAULTED;
	END_IF

	UpdateStatus;

	//Empty belt status
	tiTimeToEmpty := REAL_TO_TIME(60 * (OverVarnish.Parameters.Hw.rOPVLength + OverVarnish.Parameters.rMediaLength) / OverVarnish.Parameters.rSpeedSetPoint);
	tonEmptyBelt.IN := OverVarnish.Inputs.xTransportMoving;
	tonEmptyBelt.PT := tiTimeToEmpty;
	tonEmptyBelt();
	IF OverVarnish.Status.Comms.xModuleOk THEN
		OverVarnish.Status.xBeltEmpty := OverVarnish.Inputs.Comms.xBeltEmpty AND (tonEmptyBelt.Q OR NOT OverVarnish.Inputs.xTransportMoving);
	ELSE
		OverVarnish.Status.xBeltEmpty := (tonEmptyBelt.Q OR NOT OverVarnish.Inputs.xTransportMoving);
	END_IF

END_ACTION

ACTION UpdateStatus:

	OverVarnish.Status.Device.xTurnedOff 	:=	OverVarnish.Status.DeviceStatus=OPV_TURNED_OFF;
	OverVarnish.Status.Device.xInit			:=	OverVarnish.Status.DeviceStatus=OPV_INIT;
	OverVarnish.Status.Device.xPreparing 	:=	OverVarnish.Status.DeviceStatus=OPV_PREPARING;
	OverVarnish.Status.Device.xReady		:=	OverVarnish.Status.DeviceStatus=OPV_READY;
	OverVarnish.Status.Device.xPriming 		:=	OverVarnish.Status.DeviceStatus=OPV_PRIMING;
	OverVarnish.Status.Device.xFaulted 		:=	OverVarnish.Status.DeviceStatus=OPV_FAULTED;

END_ACTION
```

### Program Logical/ExtPack/_Ancillaries/OpvCtrl/OpvSim/OpvSim_v1/OpvSim (IEC)

#### OpvSim.var
```iecst
VAR
	SimOpv : REFERENCE TO OpvSim_typ;
	Opv : REFERENCE TO Opv_typ;
	tonTransport : TON;
	tonReady : TON;
	tonPrime : TON;
	tonBeltEmpty : TON;
	tonDry : TON;
END_VAR
```

### OpvSim.typ
```iecst
TYPE
	OPVSimCommands_typ : 	STRUCT
		CreateError : BOOL;
	END_STRUCT;
	OpvSim_typ : 	STRUCT
		Commands : OPVSimCommands_typ;
	END_STRUCT;
END_TYPE
```

### Program Logical/ExtPack/_Ancillaries/PrimerCtrl/PrimerCtrl_v1/PrimerCtrl (IEC)

#### Primer.st - Init, cyclic, exit code
```iecst
PROGRAM _CYCLIC

	Primer ACCESS ADR(gPrimer);

	//Version
	Primer.Status.Version.iVersion0 := Primer.Inputs.Comms.iVersion1;
	Primer.Status.Version.iVersion1 := Primer.Inputs.Comms.iVersion2;
	Primer.Status.Version.iVersion2 := Primer.Inputs.Comms.iVersion3;
	Primer.Status.Version.iVersion3 := Primer.Inputs.Comms.iVersion4;

	//Model evaluation
	iPrimerModel.0 := Primer.Inputs.xModelInput[0];
	iPrimerModel.1 := Primer.Inputs.xModelInput[1];
	iPrimerModel.2 := Primer.Inputs.xModelInput[2];

	Primer.Parameters.xInstalled := iPrimerModel>0;

	//Specify Type of primer Model
	Primer.Status.iModel := iPrimerModel;
	CASE iPrimerModel OF
		1: Primer.Status.PrimerType := PRIMERTY_GIARDINA;
		2: Primer.Status.PrimerType := PRIMERTY_DMS;
		3: Primer.Status.PrimerType := PRIMERTY_TECLIGHTNING;
		ELSE Primer.Status.PrimerType := PRIMERTY_UNDEFINED;
	END_CASE

	IF NOT Primer.Parameters.xInstalled OR NOT Primer.ParSw.xEnabled THEN
		ResetAlarms;
		Primer.Outputs.Physical := PhysicalOutputsReset;
		Primer.Commands:=ResetCommands;
		Primer.Status.DeviceStatus:=PRIMER_TURNED_OFF;
		CopyOfWriteData := EraseWriteData;
		Primer.Status.xBeltEmpty := TRUE;
		UpdateStatus;
		RETURN;
	END_IF

	IF Primer.Commands.xResetAlarms THEN ResetAlarms; END_IF

	Configuration;

	Status;

	IF NOT Primer.Parameters.xSimulationMode THEN
		AssignDataComms;
	END_IF

	//Erasing data when ancillary not in remote
	IF NOT Primer.Inputs.Comms.xRemote THEN
		CopyOfWriteData := EraseWriteData;
	END_IF

	Alarms;

	IF Primer.Status.Device.xFaulted OR Primer.Status.Device.xTurnedOff OR NOT Primer.Parameters.xLineInAuto THEN
		Primer.Status.CtrlStatus:=PRIMERCTRL_STOPPED;
	END_IF

	CASE Primer.Status.CtrlStatus OF
		PRIMERCTRL_STOPPED:
			//Actions
			Primer.Outputs.Physical := PhysicalOutputsReset;

			//Transition
			IF Primer.Commands.xPrepare THEN
				xEnablePriming:= Primer.ParSw.xEnablePriming AND Primer.Orders.xEnablePriming;
				Primer.Status.CtrlStatus:=PRIMERCTRL_PREPARING;
			END_IF

		PRIMERCTRL_STOPPING:
			//Actions
			Primer.Outputs.Physical := PhysicalOutputsReset;

			//Transition
			IF Primer.Status.DeviceStatus=PRIMER_TURNED_OFF OR Primer.Status.DeviceStatus=PRIMER_INIT THEN
				Primer.Status.CtrlStatus:=PRIMERCTRL_STOPPED;
			END_IF

		PRIMERCTRL_CONTROLSTOPPING:
			//Wait to have the belt empty and send the Stop order
			IF (Primer.Status.xBeltEmpty AND EDGEPOS(Primer.Orders.xDisableReadBlock)) OR NOT Primer.Inputs.xTransportMoving THEN
				Primer.Status.CtrlStatus:=PRIMERCTRL_STOPPING;
			END_IF

		PRIMERCTRL_PREPARING:
			//Actions

			IF xEnablePriming THEN
				Primer.Outputs.Physical.xRunTransport:=TRUE;
				Primer.Outputs.Physical.xPrepareToPrime:=TRUE;
				//Transition
				IF Primer.Status.DeviceStatus=PRIMER_READY THEN
					Primer.Status.CtrlStatus:=PRIMERCTRL_PREPARED;
				END_IF

			ELSE
				Primer.Outputs.Physical.xRunTransport:=TRUE;
				//Transition
				IF Primer.Status.DeviceStatus=PRIMER_BELT_RUNNING THEN
					Primer.Status.CtrlStatus:=PRIMERCTRL_PREPARED;
				END_IF

			END_IF

		PRIMERCTRL_PAUSED,
		PRIMERCTRL_PREPARED:
			//Actions
			IF Primer.Commands.xStart THEN
				Primer.Status.CtrlStatus:=PRIMERCTRL_STARTING;
			END_IF

		PRIMERCTRL_STARTING:
			//Actions
			IF xEnablePriming THEN
				Primer.Outputs.Physical.xRunPriming:=TRUE;
				IF Primer.Status.DeviceStatus=PRIMER_PRIMING THEN
					Primer.Outputs.Physical.xRunDryer:=TRUE;
				END_IF
				//Transition
				IF Primer.Status.DeviceStatus=PRIMER_DRYING THEN
					Primer.Status.CtrlStatus:=PRIMERCTRL_WORKING;
				END_IF
			ELSE
				Primer.Outputs.Physical.xRunTransport:=TRUE;
				IF Primer.Status.DeviceStatus=PRIMER_BELT_RUNNING THEN
					Primer.Status.CtrlStatus:=PRIMERCTRL_WORKING;
				END_IF
			END_IF

			//Transition
			IF Primer.Commands.xPause THEN
				Primer.Status.CtrlStatus:=PRIMERCTRL_PAUSING;
			END_IF

		PRIMERCTRL_WORKING:
			IF Primer.Commands.xPause THEN
				Primer.Status.CtrlStatus:=PRIMERCTRL_PAUSING;
			END_IF

		PRIMERCTRL_PAUSING:
			//Wait to empty the Belt to avoid media inside
			IF Primer.Status.xBeltEmpty THEN
				IF xEnablePriming THEN
					Primer.Outputs.Physical.xRunDryer:=FALSE;
					//Transition
					IF Primer.Status.DeviceStatus=PRIMER_PRIMING THEN
						Primer.Status.CtrlStatus:=PRIMERCTRL_PAUSED;
					END_IF
				ELSE
					IF Primer.Status.DeviceStatus=PRIMER_INIT OR Primer.Status.DeviceStatus=PRIMER_BELT_RUNNING THEN
						Primer.Status.CtrlStatus:=PRIMERCTRL_PAUSED;
					END_IF
				END_IF
			END_IF

	END_CASE

	IF Primer.Commands.xStop THEN
		Primer.Status.CtrlStatus:=PRIMERCTRL_STOPPING;
	ELSIF Primer.Commands.xControlStop THEN
		Primer.Status.CtrlStatus:=PRIMERCTRL_CONTROLSTOPPING;
	END_IF

	//Store the history of the status to easy the debug
	IF Primer.Status.CtrlStatus<>StateHistory[0] THEN
		FOR iIndexHistory:=iHistoryLines TO 1 BY -1 DO
			StateHistory[iIndexHistory]:=StateHistory[iIndexHistory-1];
		END_FOR
		StateHistory[0]:=Primer.Status.CtrlStatus;
	END_IF

	//Fall down the commands
	Primer.Commands:=ResetCommands;

END_PROGRAM
```

#### Configuration.st
```iecst
ACTION Configuration:

	CASE Primer.Status.PrimerType OF
		PRIMERTY_GIARDINA:
			Primer.Parameters.Hw.iMaxMediaWidth := 1800;
			Primer.Parameters.Hw.iMaxMediaLength := 3000;
			Primer.Parameters.Hw.rPrimerLength := 3000;
			Primer.Parameters.Hw.iMinMediaThickness := 8;
			Primer.Parameters.Hw.iMaxMediaThickness := 160;
			Primer.Parameters.Hw.xDoubleLineAllowed := TRUE;

		PRIMERTY_DMS:
			Primer.Parameters.Hw.iMaxMediaWidth := 1800;
			Primer.Parameters.Hw.iMaxMediaLength := 3000;
			Primer.Parameters.Hw.rPrimerLength := 3000;
			Primer.Parameters.Hw.iMinMediaThickness := 10;
			Primer.Parameters.Hw.iMaxMediaThickness := 150;
			Primer.Parameters.Hw.xDoubleLineAllowed := TRUE;

		PRIMERTY_TECLIGHTNING:
			Primer.Parameters.Hw.iMaxMediaWidth := 1800;
			Primer.Parameters.Hw.iMaxMediaLength := 3200;
			Primer.Parameters.Hw.rPrimerLength := 3000;
			Primer.Parameters.Hw.iMinMediaThickness := 3;
			Primer.Parameters.Hw.iMaxMediaThickness := 120;
			Primer.Parameters.Hw.xDoubleLineAllowed := FALSE;

	END_CASE

END_ACTION
```

#### PrimerCtrl.var - Local variables
```iecst
VAR
	Primer : REFERENCE TO Primer_typ;
	AlarmsReseted : PrimerAlarms_typ;
	ResetCommands : PrimerCommands_typ;
	xEnablePriming : BOOL; (*Active if priming is enabled from SW and from Printer/Line*)
	tiTimeToEmpty : TIME;
	tonEmptyBelt : TON;
	CommsReset : PrimerCommsInputs_typ;
	PhysicalOutputsReset : PrimerPhysicalOutputs_typ;
	iPrimerModel : USINT;
	iIndexHistory : USINT;
	StateHistory : ARRAY[0..iHistoryLines] OF PrimerCtrlStatus_enum;
END_VAR
VAR CONSTANT
	iHistoryLines : USINT := 20;
END_VAR
VAR
	rPrevWidth : REAL;
	rPrevGap : REAL;
	rPrevThickness : REAL;
	rPrevLength : REAL;
	xBoardParametersChanged : BOOL;
	tof_BoardParametersChanged : TOF;
	ModSlaveState : UINT;
	LastError : UINT;
	LastErrorBlockNum : UINT;
	CopyOfWriteData : ARRAY[1..25] OF UINT;
	tonDisableWrittingOfData : TON;
	xDisableWriteData : BOOL;
	ton_CommsError : TON;
	EraseWriteData : ARRAY[1..25] OF UINT;
END_VAR
```

### Primer.typ
```iecst
TYPE
	PrimerCtrlStatus_enum :
		(
		PRIMERCTRL_STOPPED,
		PRIMERCTRL_STOPPING,
		PRIMERCTRL_PREPARING,
		PRIMERCTRL_PREPARED,
		PRIMERCTRL_PAUSING,
		PRIMERCTRL_PAUSED,
		PRIMERCTRL_STARTING,
		PRIMERCTRL_WORKING,
		PRIMERCTRL_CONTROLSTOPPING
		);
	PrimerStatus_enum :
		(
		PRIMER_TURNED_OFF,
		PRIMER_INIT,
		PRIMER_PREPARING,
		PRIMER_READY,
		PRIMER_DRYING,
		PRIMER_FAULTED,
		PRIMER_PRIMING,
		PRIMER_BELT_RUNNING
		);
	PrimerType_enum :
		(
		PRIMERTY_UNDEFINED,
		PRIMERTY_GIARDINA,
		PRIMERTY_DMS,
		PRIMERTY_TECLIGHTNING
		);
	PrimerCommsInputs_typ : 	STRUCT
		xCommsOK : BOOL; (*Modbus communications are working properly*)
		uiTransportSpeed : UINT;
		uiCoaterRollerSpeed : UINT;
		xRemote : BOOL;
		xSpeedMode : BOOL; (*Belt empty in the device*)
		xBeltEmpty : BOOL; (*Belt empty in the device*)
		iVersion1 : INT; (*Machine platform (Nozomi = 1)*)
		iVersion2 : INT; (*Machine project (C18000 = 0 / C14000 = 1)*)
		iVersion3 : INT; (*Hardware version*)
		iVersion4 : INT; (*Sotfware version*)
		iStatus : INT; (*Status word*)
		xStopButtonPressed : BOOL;
	END_STRUCT;
	PrimerInputs_typ : 	STRUCT
		xPrimerPresent : BOOL;
		xReadyToPrime : BOOL;
		xCoating : BOOL;
		xError : BOOL;
		xCoatingLevelLow : BOOL;
		xTransportMoving : BOOL;
		xDryerInRun : BOOL;
		xCriticalAlarm : BOOL;
		iCoaterModel : INT;
		xModelInput : ARRAY[0..2]OF BOOL;
		xNoPowered : BOOL;
		Comms : PrimerCommsInputs_typ;
		xIrPowered : BOOL;
		xUvPowered : BOOL;
	END_STRUCT;
	PrimerOutputs_typ : 	STRUCT
		Physical : PrimerPhysicalOutputs_typ;
		Comms : PrimerCommsOutputs_typ;
	END_STRUCT;
	PrimerAlarms_typ : 	STRUCT
		xError : BOOL;
		xNoPrimerPresent : BOOL;
		xCoatingLevelLow : BOOL;
		xAnyAlarm : BOOL;
		xNotRemote : BOOL;
		xCoatingRecircNotEnabled : BOOL;
		xNoPowered : BOOL;
		xCriticalAlarm : BOOL;
		xWarningAlarm : BOOL;
		xCommsError : BOOL;
		xStopRequest : BOOL; (*Stop request from Dryer when physical stop button is pressed*)
	END_STRUCT;
	PrimerParametersSw_typ : 	STRUCT
		xEnabled : BOOL; (*This variable replaces the previous "xThereIs". Activated by SW*)
		xEnablePriming : BOOL; (*Priming enabled from SW*)
	END_STRUCT;
	PrimerParametersHw_typ : 	STRUCT
		iMaxMediaWidth : UINT; (*Maximum media width allowed in mm*)
		iMinMediaWidth : UINT; (*Minimum media width allowed in mm*)
		iMaxMediaLength : UINT; (*Maximum media length allowed in mm*)
		iMinMediaLength : UINT; (*Minimum media length allowed in mm*)
		rPrimerLength : REAL; (*Length in mm*)
		rMaxSpeed : REAL := 100.0; (*Maximum speed allowed in m/min*)
		iMinMediaThickness : UINT; (*Minimum media height allowed in tenth of mm*)
		iMaxMediaThickness : UINT; (*Maximum media height allowed in tenth of mm*)
		xDoubleLineAllowed : BOOL; (*Active when printer allows double line printing*)
	END_STRUCT;
	PrimerParameters_typ : 	STRUCT
		xInstalled : BOOL;
		xSimulationMode : BOOL; (*Defined by the configuration in Automation Studio*)
		xAlrPresent : BOOL;
		xLineInAuto : BOOL;
		xPreviousDeviceStopped : BOOL; (*Length in mm*)
		rMediaLength : REAL; (*Length in mm*)
		rSpeedSetPoint : REAL; (*Speed in m/min*)
		Media : PrimerMediaParameters;
		rLineAccelRate : REAL := 2; (*mm/s2 (2.5m/s2*60=150mpm/s)*)
		rLineDecelRate : REAL := 2; (*mm/s2 (2.5m/s2*60=150mpm/s)*)
		rBeltSpeedSetPoint : REAL;
		xDoubleLine : BOOL;
		LineState : LineStatus_enum;
		LineStatusSummary : LineControlStatusSummarized;
		Hw : PrimerParametersHw_typ;
		xActiveSlaveDiagnosis : BOOL;
	END_STRUCT;
	PrimerCommands_typ : 	STRUCT
		xStart : BOOL; (*Edge commands. Reseted when managed*)
		xPrepare : BOOL; (*Edge commands. Reseted when managed*)
		xPause : BOOL; (*Edge commands. Reseted when managed*)
		xBelEmpty : BOOL; (*Edge commands. Reseted when managed*)
		xControlStop : BOOL; (*Edge commands. Reseted when managed*)
		xStop : BOOL; (*Edge commands. Reseted when managed*)
		xThereIsPrimer : BOOL;
		xResetAlarms : BOOL;
		xEnteringMedia : BOOL;
		xNewBoardParameters : BOOL; (*Pulse to let know board paramters have changed*)
	END_STRUCT;
	PrimerDeviceStatus_typ : 	STRUCT
		xTurnedOff : BOOL;
		xInit : BOOL;
		xPreparing : BOOL;
		xEmpty : BOOL;
		xReady : BOOL;
		xPriming : BOOL;
		xDrying : BOOL;
		xFaulted : BOOL;
	END_STRUCT;
	PrimerStatus_typ : 	STRUCT
		iModel : USINT; (*Model of the Device. 0:Retroflex*)
		Version : EFI_version_typ;
		CtrlStatus : PrimerCtrlStatus_enum;
		DeviceStatus : PrimerStatus_enum;
		Device : PrimerDeviceStatus_typ;
		xBeltEmpty : BOOL;
		PrimerType : PrimerType_enum;
		Comms : PrimerCommsStatus_typ;
	END_STRUCT;
	Primer_typ : 	STRUCT
		Inputs : PrimerInputs_typ;
		Outputs : PrimerOutputs_typ;
		Alarms : PrimerAlarms_typ;
		ParSw : PrimerParametersSw_typ;
		Parameters : PrimerParameters_typ;
		Commands : PrimerCommands_typ;
		Status : PrimerStatus_typ;
		Orders : PrimerOrders_typ;
	END_STRUCT;
	PrimerPhysicalOutputs_typ : 	STRUCT
		xPrepareToPrime : BOOL;
		xRunPriming : BOOL;
		xRunTransport : BOOL;
		xRunDryer : BOOL;
	END_STRUCT;
	PrimerCommsOutputs_typ : 	STRUCT
		iControl : UINT; (*Status word*)
		iControl2 : UINT; (*Status word*)
	END_STRUCT;
	PrimerMediaParameters : 	STRUCT
		rThickness : REAL; (*Tile thickness to print from gui in mm*)
		rWidth : REAL; (*Board's width in mm*)
		rGap : REAL; (*Gap between boards in mm*)
		rLength : REAL; (*Board's length in mm*)
		rOffsetRegisterL1 : REAL; (*Board's width in mm*)
		rOffsetRegisterL2 : REAL; (*Board's width in mm*)
	END_STRUCT;
	PrimerCommsStatus_typ : 	STRUCT
		xModuleOk : BOOL;
		ModSlaveState : UINT;
		LastError : UINT;
		LastErrorBlockNum : UINT;
		xStopButtonPressed : BOOL;
		ActOverloadError : BOOL;
		ActModbusError : BOOL;
		ActSlvConError : BOOL;
		ActRefreshError : BOOL;
		ActInternalError : BOOL;
		ActConfError : BOOL;
		HistOverloadError : BOOL;
		HistModbusError : BOOL;
		HistSlvConError : BOOL;
		HistRefreshError : BOOL;
		HistInternalError : BOOL;
		HistConfError : BOOL;
		ModbusErrorCnt : UINT;
		ModbusConErrorCnt : UINT;
		ModbusPktRefreshTimeoutCnt : UINT;
		ModbusPktPendPerSec : UINT;
		ModbusMeanResponseTime : UINT;
	END_STRUCT;
	PrimerOrders_typ : 	STRUCT
		xDisableWriteBlock : BOOL;
		xDisableReadBlock : BOOL;
		xEnablePriming : BOOL; (*Priming enabled from printer/line*)
	END_STRUCT;
END_TYPE
```

### Sarm.typ
```iecst
TYPE
	SarmCtrlStatus_enum :
		(
		SARMCTRL_STOPPED,
		SARMCTRL_STOPPING,
		SARMCTRL_STARTING,
		SARMCTRL_RUNNING,
		SARMCTRL_PAUSING,
		SARMCTRL_PAUSED,
		SARMCTRL_CONTROLSTOPPING
		);
	SarmStatus_enum :
		(
		Sarm_TURNED_OFF,
		Sarm_INIT,
		Sarm_PREPARING,
		Sarm_READY,
		Sarm_FAKESTATE,
		Sarm_FAULTED
		);
	SarmType_enum :
		(
		SARMTY_UNDEFINED,
		SARMTY_V1
		);
	SarmInputs_typ : 	STRUCT
		xRunning : BOOL;
		xError : BOOL;
		xModelInput : ARRAY[0..2]OF BOOL;
		xPowered : BOOL;
		xSarmPresent : BOOL;
		Comms : SarmCommsInputs_typ;
	END_STRUCT;
	SarmOutputs_typ : 	STRUCT
		xFastStop : BOOL;
		xStartTransport : BOOL;
		Comms : SarmCommsOutputs_typ;
	END_STRUCT;
	SarmAlarms_typ : 	STRUCT
		xError : BOOL;
		xNotRemote : BOOL;
		xAnyAlarm : BOOL;
		xNoPowered : BOOL;
		xCriticalAlarm : BOOL;
		xWarningAlarm : BOOL;
		xCommsError : BOOL;
	END_STRUCT;
	SarmParametersSw_typ : 	STRUCT
		xEnabled : BOOL;
		xBatchFeeding : BOOL; (*1:Batch feeding mode; 0: continuous feeding.*)
		iCentralOffset : INT; (*Offset value received from SW for Sarms with Parameters.Hw.xOffsetAvailable = TRUE;*)
	END_STRUCT;
	SarmParametersHw_typ : 	STRUCT
		iMaxMediaWidth : UINT; (*Maximum media width allowed in mm*)
		iMinMediaWidth : UINT; (*Minimum media width allowed in mm*)
		iMinMediaLength : UINT; (*Minimum media length allowed in mm*)
		iMaxMediaLength : UINT; (*Maximum media length allowed in mm*)
		iMaxOffset : UINT; (*Upper limit for line alignment offset value [mm]*)
		iMinOffset : INT; (*Lower limit for line alignment offset value [mm]*)
		iMinMediaThickness : UINT; (*Minimum media height allowed in tenth of mm*)
		iMaxMediaThickness : UINT; (*Maximum media height allowed in tenth of mm*)
		rSarmLength : REAL; (*Length in mm*)
		rMaxSpeed : REAL := 60.0; (*Maximum speed allowed in m/min*)
		xDoubleLineAllowed : BOOL; (*Active when allows double line printing*)
	END_STRUCT;
	SarmParameters_typ : 	STRUCT
		xInstalled : BOOL;
		xSimulationMode : BOOL; (*Defined by the configuration in Automation Studio*)
		xCommsOK : BOOL;
		LineState : LineStatus_enum;
		xLineInAuto : BOOL;
		Media : SarmMediaParameters;
		xDoubleLine : BOOL;
		Hw : SarmParametersHw_typ;
		xActiveSlaveDiagnosis : BOOL;
		xPreviousDeviceEmpty : BOOL;
		rMediaLength : REAL; (*Length in mm*)
		rSpeedSetPoint : REAL; (*Speed in m/min*)
		iLineConfig : UINT;
	END_STRUCT;
	SarmCommands_typ : 	STRUCT
		xBelEmpty : BOOL; (*Edge commands. Reseted when managed*)
		xStart : BOOL; (*Edge commands. Reseted when managed*)
		xPause : BOOL; (*Edge commands. Reseted when managed*)
		xControlStop : BOOL; (*Edge commands. Reseted when managed*)
		xStop : BOOL; (*Edge commands. Reseted when managed*)
		xResetAlarms : BOOL;
		xNewBoardParameters : BOOL; (*Set 1 when there is sent a new configuration.*)
		xNewOrder : BOOL; (*New batch. Set when there is sent a new job. This signal reset the current counter*)
	END_STRUCT;
	SarmDeviceStatus_typ : 	STRUCT
		xTurnedOff : BOOL;
		xInit : BOOL;
		xPreparing : BOOL;
		xReady : BOOL;
		xFaulted : BOOL;
	END_STRUCT;
	SarmStatus_typ : 	STRUCT
		iModel : USINT := 1; (*Model of the Device*)
		Version : EFI_version_typ;
		CtrlStatus : SarmCtrlStatus_enum;
		DeviceStatus : SarmStatus_enum;
		Device : SarmDeviceStatus_typ;
		SarmType : SarmType_enum;
		Comms : SarmCommsStatus_typ;
		xInstalled : BOOL;
		xBeltEmpty : BOOL;
	END_STRUCT;
	Sarm_typ : 	STRUCT
		Inputs : SarmInputs_typ;
		Outputs : SarmOutputs_typ;
		Alarms : SarmAlarms_typ;
		ParSw : SarmParametersSw_typ;
		Parameters : SarmParameters_typ;
		Commands : SarmCommands_typ;
		Status : SarmStatus_typ;
		Orders : SarmOrders_typ;
	END_STRUCT;
	SarmCommsOutputs_typ : 	STRUCT
		iControl : INT; (*Status word*)
	END_STRUCT;
	SarmCommsInputs_typ : 	STRUCT
		xSafetyOnline : BOOL;
		xOnline : BOOL; (*Recirculation of the Sarm enabled in the device*)
		xPositionReady : BOOL; (*Recirculation of the Sarm enabled in the device*)
		xWarningPresent : BOOL; (*Recirculation of the Sarm enabled in the device*)
		xAlarmPresent : BOOL; (*Recirculation of the Sarm enabled in the device*)
		xRemote : BOOL; (*Recirculation of the Sarm enabled in the device*)
		xBeltEmpty : BOOL;
		iVersion1 : INT; (*Machine platform (Nozomi = 1)*)
		iVersion2 : INT; (*Machine project (C18000 = 0 / C14000 = 1)*)
		iVersion3 : INT; (*Hardware version*)
		iVersion4 : INT; (*Sotfware version*)
		iStatus : INT; (*Status word*)
		iAlarmWord1 : INT; (*Status word*)
		iAlarmWord2 : INT; (*Status word*)
		iAlarmWord3 : INT; (*Status word*)
	END_STRUCT;
	SarmMediaParameters : 	STRUCT
		rThickness : REAL; (*Tile thickness to print from gui in mm*)
		rWidth : REAL; (*Board's width in mm*)
		rGap : REAL; (*Gap between boards in mm*)
		rLength : REAL; (*Board's length in mm*)
		rOffsetRegisterL1 : REAL; (*Board's width in mm*)
		rOffsetRegisterL2 : REAL; (*Board's width in mm*)
	END_STRUCT;
	SarmCommsStatus_typ : 	STRUCT
		xModuleOk : BOOL;
		ModSlaveState : UINT;
		LastError : UINT;
		LastErrorBlockNum : UINT;
		xStopButtonPressed : BOOL;
		ActOverloadError : BOOL;
		ActModbusError : BOOL;
		ActSlvConError : BOOL;
		ActRefreshError : BOOL;
		ActInternalError : BOOL;
		ActConfError : BOOL;
		HistOverloadError : BOOL;
		HistModbusError : BOOL;
		HistSlvConError : BOOL;
		HistRefreshError : BOOL;
		HistInternalError : BOOL;
		HistConfError : BOOL;
		ModbusErrorCnt : UINT;
		ModbusConErrorCnt : UINT;
		ModbusPktRefreshTimeoutCnt : UINT;
		ModbusPktPendPerSec : UINT;
		ModbusMeanResponseTime : UINT;
		xBeltEmpty : BOOL;
	END_STRUCT;
	SarmOrders_typ : 	STRUCT
		xDisableReadBlock : BOOL;
		xDisableWriteBlock : BOOL;
	END_STRUCT;
END_TYPE
```

### Program Logical/ExtPack/_Ancillaries/SarmCtrl/SarmCtrl/SarmCtrl

#### SarmCtrl.var
```iecst
VAR
	Sarm : REFERENCE TO Sarm_typ;
	AlarmsReseted : SarmAlarms_typ;
	ResetCommands : SarmCommands_typ;
	CommsReset : SarmCommsInputs_typ;
	OutputsReset : SarmOutputs_typ;
	iSarmModel : USINT;
	iIndexHistory : USINT;
	StateHistory : ARRAY[0..iHistoryLines] OF SarmCtrlStatus_enum;
END_VAR
VAR CONSTANT
	iHistoryLines : USINT := 20;
END_VAR
VAR
	ModSlaveState : UINT;
	LastError : UINT;
	LastErrorBlockNum : UINT;
	tiTimeToEmpty : TIME;
	tonEmptyBelt : TON;
	EraseWriteData : ARRAY[1..25] OF UINT;
	CopyOfWriteData : ARRAY[1..25] OF UINT;
	tonDisableWrittingOfData : TON;
	xDisableWriteData : BOOL;
	ton_CommsError : TON;
END_VAR
```

#### Alarms.st
```iecst
ACTION Alarms:

	//Sarm No Powered Warning
	IF NOT Sarm.Inputs.xPowered THEN Sarm.Alarms.xNoPowered := TRUE; END_IF

	IF Sarm.Inputs.xError THEN
		Sarm.Alarms.xError := TRUE;
	END_IF

	//Saving modbus slave status when comms error raises
	IF EDGEPOS (Sarm.Alarms.xCommsError) THEN
		ModSlaveState := Sarm.Status.Comms.ModSlaveState;
		LastError := Sarm.Status.Comms.LastError;
		LastErrorBlockNum := Sarm.Status.Comms.LastErrorBlockNum;
	END_IF

	//Alarms related to comms
	IF Sarm.Status.Comms.xModuleOk THEN
		//Remote
		IF (NOT Sarm.Inputs.Comms.xRemote) AND Sarm.Parameters.xLineInAuto THEN
			Sarm.Alarms.xNotRemote := TRUE;
		END_IF
	END_IF

	//Data write to ancillaries is critical to be updated properly. So just write block is monitored to raise comms alarm
	//Added ancillary first command used to get it ready to check comms also.
	//Read function not considered as the only variable critical for line process is to acknowledge "belt empty" status and in case of module nOk
	//timer "tonEmptyBelt" is executed
	ton_CommsError.IN := NOT Sarm.Status.Comms.xModuleOk AND (NOT Sarm.Orders.xDisableWriteBlock OR Sarm.Commands.xStart);
	ton_CommsError.PT := T#500ms;
	ton_CommsError();

	IF ton_CommsError.Q  THEN
		Sarm.Alarms.xCommsError := TRUE;
	END_IF

	//Alarms Summary
	//Critical
	Sarm.Alarms.xCriticalAlarm:=	Sarm.Alarms.xError OR
									Sarm.Alarms.xNoPowered OR
									Sarm.Alarms.xNotRemote OR
									Sarm.Alarms.xCommsError;

	//Warning
	//Sarm.Alarms.xWarningAlarm	:=	;

END_ACTION

ACTION ResetAlarms:
	Sarm.Alarms := AlarmsReseted;
END_ACTION
```

### SarmSim.var
```iecst
VAR
	SimSarm : REFERENCE TO SarmSim_typ;
	Sarm : REFERENCE TO Sarm_typ;
	tonPrepare : TON;
END_VAR
```

### Program Logical/ExtPack/_Ancillaries/StackerCtrl/StackerCtrl_v1/StackerCtrl (IEC)

#### Alarms.st
```iecst
ACTION Alarms:

	Stacker.Alarms.xNoStackerPresent:= NOT Stacker.Inputs.xStackerPresent;

	//Related to physical inputs
	//If no Stacker, define that alarm and exit
	IF Stacker.Alarms.xNoStackerPresent THEN
		ResetAlarms;
		Stacker.Alarms.xNoStackerPresent:=TRUE;
	END_IF

	//No Powered
	IF Stacker.Inputs.xNoPowered THEN Stacker.Alarms.xNoPowered := TRUE; END_IF

	//Error
	IF Stacker.Inputs.xError THEN
		Stacker.Alarms.xError := TRUE;
	END_IF

	//Stacker not running (DELOREAN-1969)
	IF xBeltsAreStopped THEN Stacker.Alarms.xBeltsStopped := TRUE; END_IF

	//Saving modbus slave status when comms error raises
	IF EDGEPOS (Stacker.Alarms.xCommsError) THEN
		ModSlaveState := Stacker.Status.Comms.ModSlaveState;
		LastError := Stacker.Status.Comms.LastError;
		LastErrorBlockNum := Stacker.Status.Comms.LastErrorBlockNum;
	END_IF

	//Alarms related to comms
	IF Stacker.Status.Comms.xModuleOk THEN
		IF (NOT Stacker.Inputs.Comms.xRemote) AND Stacker.Parameters.xLineInAuto THEN
			Stacker.Alarms.xNotRemote := TRUE;
		END_IF
	END_IF

	//Data write to ancillaries is critical to be updated properly. So just write block is monitored to raise comms alarm
	//Added ancillary first command used to get it ready to check comms also.
	//Read function not considered as the only variable critical for line process is to acknowledge "belt empty" status and in case of module nOk
	//timer "tonEmptyBelt" is executed
	ton_CommsError.IN := NOT Stacker.Status.Comms.xModuleOk AND (NOT Stacker.Orders.xDisableWriteBlock OR Stacker.Commands.xPrepare);
	ton_CommsError.PT := T#500ms;
	ton_CommsError();

	IF ton_CommsError.Q  THEN
		Stacker.Alarms.xCommsError := TRUE;
	END_IF

	//General
	IF (Stacker.Orders.xRejectSheet OR Stacker.Orders.xHoldReject) AND NOT Stacker.Inputs.Comms.xRejectAvailable THEN
		Stacker.Alarms.xRejectNoAvailable := TRUE;
	END_IF

	//Alarms Summary
	//Critical
	Stacker.Alarms.xCriticalAlarm:= 	Stacker.Alarms.xError OR
										Stacker.Alarms.xNoPowered OR
										Stacker.Alarms.xNotRemote OR
										Stacker.Alarms.xBeltsStopped OR
										Stacker.Alarms.xCommsError;
	//Warning
	Stacker.Alarms.xWarningAlarm	:=	Stacker.Alarms.xRejectNoAvailable;

END_ACTION

ACTION ResetAlarms:
	Stacker.Alarms := AlarmsReseted;
END_ACTION
```

#### AssignDataComms.st
```iecst
ACTION AssignDataComms:

	//Active modbus slave diagnosis when ancillary is enabled. This parameter must remain to TRUE from then on.
	//Just would be set to FALSE via UaExpert, to reset historic errors when ancillary is disabled
	Stacker.Parameters.xActiveSlaveDiagnosis := TRUE;

	/////////////////
	//Pre bits treatment
	Stacker.Comms.iControl.0 := Stacker.Comms.xEndCycle;
	Stacker.Comms.iControl.1 := Stacker.Comms.xCleanBelts := Stacker.Outputs.xCleanBelts;
	Stacker.Comms.iControl.2 := Stacker.Comms.xResetAlarms;
	Stacker.Comms.iControl.3 := Stacker.ParSw.xStackMode;
	Stacker.Comms.iControl.4 := Stacker.Comms.xLastBox;
	Stacker.Comms.iControl.5 := Stacker.Orders.xHoldReject;
	Stacker.Comms.iControl.6 := Stacker.Parameters.xDoubleLine;

	//Write Registers
	gToWriteDataModbStacker[1] := Stacker.Comms.iControl;
	gToWriteDataModbStacker[2] := REAL_TO_UINT(Stacker.Parameters.Media.rLength*10);
	gToWriteDataModbStacker[3] := REAL_TO_UINT(Stacker.Parameters.Media.rWidth*10);
	gToWriteDataModbStacker[4] := REAL_TO_UINT(Stacker.Parameters.Media.rThickness*10);
	gToWriteDataModbStacker[5] := REAL_TO_UINT(Stacker.Parameters.Media.rGap*10);
	gToWriteDataModbStacker[6] := Stacker.ParSw.iStackBoardsNum;
	gToWriteDataModbStacker[7] := Stacker.ParSw.iStackHeight;
	gToWriteDataModbStacker[8] := REAL_TO_UINT(Stacker.Parameters.rSpeedSetPoint*10);
	(*gToWriteDataModbStacker[9] := ;
	gToWriteDataModbStacker[10] := ;
	gToWriteDataModbStacker[11] := ;

	gToWriteDataModbStacker[12] := ;
	gToWriteDataModbStacker[13] := ;
	gToWriteDataModbStacker[14] := ;
	gToWriteDataModbStacker[15] := ;
	gToWriteDataModbStacker[16] := ;
	gToWriteDataModbStacker[17] := ;
	gToWriteDataModbStacker[18] := ;
	gToWriteDataModbStacker[19] := ;
	gToWriteDataModbStacker[20] := ;
	gToWriteDataModbStacker[21] := ;
	gToWriteDataModbStacker[22] := ;
	gToWriteDataModbStacker[23] := ;
	gToWriteDataModbStacker[24] := ;
	gToWriteDataModbStacker[25] := ;
	*)

	//Disabling writting after some time active. To test
	tonDisableWrittingOfData.IN:= NOT xDisableWriteData;
	tonDisableWrittingOfData.PT:= T#1000ms;
	tonDisableWrittingOfData();

	IF tonDisableWrittingOfData.Q THEN
		xDisableWriteData := TRUE;
	END_IF

	FOR iIndex:=1 TO 25 DO
		IF gToWriteDataModbStacker[iIndex]<>CopyOfWriteData[iIndex] THEN
			xDisableWriteData := FALSE;
		END_IF
	END_FOR

	Stacker.Orders.xDisableWriteBlock := xDisableWriteData;

	//Copying previous data
	CopyOfWriteData := gToWriteDataModbStacker;

	////////////////
	//Read Registers
	IF Stacker.Status.Comms.xModuleOk THEN
		Stacker.Inputs.Comms.iStatus := gReceivedDataModbStacker[1];
		Stacker.Inputs.Comms.uiNumBoardsInCurrentPile := gReceivedDataModbStacker[2];
		Stacker.Inputs.Comms.uiCurrentPileHeigh := gReceivedDataModbStacker[3];
		Stacker.Inputs.Comms.uiTransportSpeed := gReceivedDataModbStacker[4];
		Stacker.Inputs.Comms.iAlarmWord1 := gReceivedDataModbStacker[5];
		Stacker.Inputs.Comms.iAlarmWord2 := gReceivedDataModbStacker[6];
		Stacker.Inputs.Comms.iAlarmWord3 := gReceivedDataModbStacker[7];
		Stacker.Inputs.Comms.iAlarmWord4 := gReceivedDataModbStacker[8];
		Stacker.Inputs.Comms.iAlarmWord5 := gReceivedDataModbStacker[9];
		Stacker.Inputs.Comms.iAlarmWord6 := gReceivedDataModbStacker[10];
		Stacker.Inputs.Comms.iAlarmWord7 := gReceivedDataModbStacker[11];
		Stacker.Inputs.Comms.iAlarmWord8:= gReceivedDataModbStacker[12];
		Stacker.Inputs.Comms.iAlarmWord9:= gReceivedDataModbStacker[13];
		Stacker.Inputs.Comms.iAlarmWord10:= gReceivedDataModbStacker[14];
		// := gReceivedDataModbStacker[15];
		// := gReceivedDataModbStacker[16];
		// := gReceivedDataModbStacker[17];
		// := gReceivedDataModbStacker[18];

		//:= gReceivedDataModbStacker[19];
		//:= gReceivedDataModbStacker[20];

		// := gReceivedDataModbStacker[21];
		Stacker.Inputs.Comms.iVersion1 := gReceivedDataModbStacker[22];
		Stacker.Inputs.Comms.iVersion2 := gReceivedDataModbStacker[23];
		Stacker.Inputs.Comms.iVersion3 := gReceivedDataModbStacker[24];
		Stacker.Inputs.Comms.iVersion4 := gReceivedDataModbStacker[25];

	END_IF

	//Post bit treatment

	Stacker.Inputs.Comms.xRemote := Stacker.Inputs.Comms.iStatus.0;
	Stacker.Inputs.Comms.xErrorActive := Stacker.Inputs.Comms.iStatus.1;
	Stacker.Inputs.Comms.xInWorkingPosition := Stacker.Inputs.Comms.iStatus.2;
	Stacker.Inputs.Comms.xStackReady := Stacker.Inputs.Comms.iStatus.3;
	Stacker.Inputs.Comms.xStackExit := Stacker.Inputs.Comms.iStatus.4;
	Stacker.Inputs.Comms.xStopDemand := Stacker.Inputs.Comms.iStatus.5;
	Stacker.Inputs.Comms.xStackerEmpty := Stacker.Inputs.Comms.iStatus.6;
	Stacker.Inputs.Comms.xBeltsEmpty := Stacker.Inputs.Comms.iStatus.7;
	Stacker.Inputs.Comms.xNewFormat := Stacker.Inputs.Comms.iStatus.8;
	Stacker.Inputs.Comms.xOnline := Stacker.Inputs.Comms.iStatus.9;
	Stacker.Inputs.Comms.xSerie := Stacker.Inputs.Comms.iStatus.10; //Serie A or B. Just make sense for full stacker
	Stacker.Inputs.Comms.xWarningActive := Stacker.Inputs.Comms.iStatus.11;
	Stacker.Inputs.Comms.xEmergencyStopNotAcknowledged := Stacker.Inputs.Comms.iStatus.12;
	Stacker.Inputs.Comms.xRejectAvailable := Stacker.Inputs.Comms.iStatus.13;

END_ACTION
```

#### Configuration.st
```iecst
ACTION Configuration:

	rMediaThickness := MAX(0, Stacker.Parameters.Media.rThickness);

	CASE Stacker.Status.StackerType OF

		STACKERTY_FULL_S:

			Stacker.Parameters.Hw.rStackerLength := 15000;

			//Media
			Stacker.Parameters.Hw.iMaxMediaWidth := 1800;
			Stacker.Parameters.Hw.iMaxMediaLength := 3000;
			Stacker.Parameters.Hw.iMinMediaThickness := 10;
			Stacker.Parameters.Hw.iMaxMediaThickness := 120;
			Stacker.Parameters.Hw.xDoubleLineAllowed := TRUE;

			//Stack
			Stacker.Parameters.Hw.iMinStackHeight := REAL_TO_UINT(iMinStackBoards*rMediaThickness);
			Stacker.Parameters.Hw.iMaxStackHeight := 1800;

			Stacker.Parameters.Hw.iMinStackBoards := 15;
			Stacker.Parameters.Hw.iMaxStackBoards := REAL_TO_UINT(UINT_TO_REAL(Stacker.Parameters.Hw.iMaxStackHeight)/rMediaThickness);

			//Reject
			Stacker.Parameters.Hw.xThereIsReject := TRUE;
			Stacker.Parameters.Hw.xRejectEjectionAvailable := TRUE;
			Stacker.Parameters.Hw.iRejectAdjustmentDistance := 12;
			Stacker.Parameters.Hw.iDistanceToReject := 230; //Measured in SN3 while debugging

		STACKERTY_BUNDLE_S:

			Stacker.Parameters.Hw.rStackerLength := 10000;

			//Media
			Stacker.Parameters.Hw.iMaxMediaWidth := 1670;
			Stacker.Parameters.Hw.iMaxMediaLength := 2440;
			Stacker.Parameters.Hw.iMinMediaThickness := 8;
			Stacker.Parameters.Hw.iMaxMediaThickness := 160;
			Stacker.Parameters.Hw.xDoubleLineAllowed := TRUE;

			//Stack
			Stacker.Parameters.Hw.iMinStackHeight := REAL_TO_UINT(iMinStackBoards*rMediaThickness);
			Stacker.Parameters.Hw.iMaxStackHeight := 300;
			Stacker.Parameters.Hw.iMinStackBoards := 15;
			Stacker.Parameters.Hw.iMaxStackBoards := REAL_TO_UINT(UINT_TO_REAL(Stacker.Parameters.Hw.iMaxStackHeight)/rMediaThickness);

			//Reject
			Stacker.Parameters.Hw.xThereIsReject := TRUE;
			Stacker.Parameters.Hw.xRejectEjectionAvailable := FALSE;
			Stacker.Parameters.Hw.iRejectAdjustmentDistance := 0;
			Stacker.Parameters.Hw.iDistanceToReject := 0; //TBD: Pending to debug in bundle stacker

	END_CASE

END_ACTION
```
